// TIA Portal V19 program export: 1 tag tables, 127 data types, 0 data blocks, 65 code blocks (in call order from the OBs), 0 instance data blocks

VAR_GLOBAL   // PLC tag table "Parameterwaardes"
END_VAR
VAR_GLOBAL CONSTANT   // user constants
   Ja : USInt := 11;
   Aan : USInt := 12;
   Open : USInt := 13;
   Beschikbaar : USInt := 14;
   InDienst : USInt := 16;
   Bevestiging : USInt := 17;
   OK : USInt := 18;
   Geactiveerd : USInt := 19;
   Auto : USInt := 128;
   Manueel : USInt := 129;
   Hand : USInt := 130;
   Sensorregeling : USInt := 112;
   Uit : USInt := 42;
   Bereikt : USInt := 15;
   Beperkt : USInt := 21;
   Gedeeltelijk : USInt := 22;
   InTransitie : USInt := 23;
   OpenVerlaten : USInt := 24;
   DeelsAfgesloten : USInt := 25;
   Onbepaald : USInt := 26;
   Nee : USInt := 41;
   Dicht : USInt := 43;
   NietBeschikbaar : USInt := 44;
   Storing : USInt := 45;
   OnvoorwaardelijkDicht : USInt := 46;
   Geen : USInt := 47;
   UitDienst : USInt := 48;
   Annulering : USInt := 49;
   Fout : USInt := 50;
   NietBereikt : USInt := 51;
   Onderdrukt : USInt := 52;
   Stop : USInt := 53;
   Overbrugd : USInt := 54;
   NOK : USInt := 55;
   Gedeactiveerd : USInt := 56;
   Gedoofd : USInt := 61;
   Rood : USInt := 62;
   GeelKnipper : USInt := 63;
   Geel : USInt := 64;
   Groen : USInt := 65;
   Leeg : USInt := 70;
   LLW : USInt := 71;
   LW : USInt := 72;
   SW : USInt := 73;
   MSW : USInt := 74;
   LHW : USInt := 75;
   HHW : USInt := 76;
   Rijrichting : USInt := 81;
   Hoog : USInt := 82;
   Max : USInt := 83;
   Gent : USInt := 84;
   Oplopend : USInt := 85;
   Dag : USInt := 86;
   Tegenrij : USInt := 91;
   Laag : USInt := 92;
   Min : USInt := 93;
   Luik : USInt := 94;
   Aflopend : USInt := 95;
   Nacht : USInt := 96;
   Lokaal : USInt := 101;
   Centraal : USInt := 102;
   Licht : USInt := 105;
   Matig : USInt := 106;
   Waarneembaar : USInt := 107;
   Ernstig : USInt := 108;
   Regeling : USInt := 111;
   Windmeting : USInt := 113;
   Bewaken : USInt := 115;
   Blussen : USInt := 116;
   Testen : USInt := 117;
   Klein : USInt := 120;
   Groot : USInt := 121;
   NietSel : USInt := 125;
   SelHand : USInt := 126;
   SelAuto : USInt := 127;
   Reset : USInt := 135;
   Parallel : USInt := 137;
   Eiland : USInt := 138;
   Live : USInt := 140;
   Boodschap : USInt := 141;
   Radio : USInt := 142;
   Gesprek : USInt := 145;
   Wacht : USInt := 146;
   Aanvraag : USInt := 147;
   Recirculatie : USInt := 150;
   Bergen : USInt := 153;
   LeegHouden : USInt := 154;
   Lozen : USInt := 155;
   OnderWater : USInt := 157;
   BovenWater : USInt := 158;
   Onderhoud : USInt := 160;
   Normaal : USInt := 161;
   Calamiteit : USInt := 162;
   StandBy : USInt := 163;
   Ondersteunend : USInt := 164;
   Evacuatie : USInt := 165;
   Vlucht : USInt := 166;
   Brand : USInt := 167;
   Waarschuw : USInt := 168;
   "TSCT+GL" : USInt := 200;   // Tunnelkoker van Gent naar Luik
   "TSCT+LG" : USInt := 201;   // Tunnelkoker van Luik naar Gent
   "TOKA+BR" : USInt := 202;   // Tunnelkoker van Brussel naar Rotterdam
   "TOKA+RB" : USInt := 203;   // Tunnelkoker van Rotterdam naar Brussel
   "TLUC+AR" : USInt := 204;   // Tunnelkoker van Antwerpen naar Rotterdam
   "TLUC+BA" : USInt := 205;   // Tunnelkoker van Brussel naar Antwerpen
   "TLUC+BR" : USInt := 206;   // Tunnelkoker van Brussel naar Rotterdam
   "TLUC+RA" : USInt := 207;   // Tunnelkoker van Rotterdam naar Antwerpen
   "TLUC+RB" : USInt := 208;   // Tunnelkoker van Rotterdam naar Brussel
   "TLUC+AB" : USInt := 209;   // Tunnelkoker van Antwerpen naar Brussel
   "TKZO+GR" : USInt := 210;   // Tunnelkoker van Gent naar Rotterdam
   "TKZO+RG" : USInt := 211;   // Tunnelkoker van Rotterdam naar Gent
   "TKZB+LG" : USInt := 212;   // Tunnelkoker van Luik naar Gent
   "TKZB+GL" : USInt := 213;   // Tunnelkoker van Gent naar Luik
   "TSCH+BR" : USInt := 214;   // Tunnelkoker van Brussel naar Rotterdam
   "TSCH+RB" : USInt := 215;   // Tunnelkoker van Rotterdam naar Brussel
   "TKZO+RA" : USInt := 216;   // Uitrit van Rotterdam naar Antwerpen
   "TKZO+AR" : USInt := 217;   // Inrit van Antwerpen naar Rotterdam
   "TKZB+KA" : USInt := 218;   // Uitrit kanalzone knooppunt naar Antwerpen
   "TKZB+LK" : USInt := 219;   // Uitrit luik naar kanaalzone knooppunt
   "TKZB+AK" : USInt := 220;   // Inrit antwerpen naar kanaalzone knooppunt
   "TKZB+KL" : USInt := 221;   // Inrit kanaalzone knooppunt naar Luik
END_VAR

TYPE "C205_VAR_IF_GVL_TYPIC"
   STRUCT
      BMO_AAN { ExternalAccessible := 'False'; ExternalVisible := 'False'; ExternalWritable := 'False'} : Bool;   // Geleideverlichting aan
      EXT_AUT { ExternalAccessible := 'False'; ExternalVisible := 'False'; ExternalWritable := 'False'} : Bool;   // Externe (hoofd) beveiliging aangesproken
      EXT_HW { ExternalAccessible := 'False'; ExternalVisible := 'False'; ExternalWritable := 'False'} : Bool;   // Sturings hardware (PLC) in storing
      STO { ExternalAccessible := 'False'; ExternalVisible := 'False'; ExternalWritable := 'False'} : Struct   // Opsomming van alle storingen en meldingen
         A001 : Bool;   // Beveiliging aangesproken
         A002 : Bool;   // Storing voeding geleideverlichting
         AT01 : Bool;   // Foute terugmelding: Geleideverlichting aangestuurd, terugmelding Aan niet (of te laat) ontvangen
         AT02 : Bool;   // Foute terugmelding: Geleideverlichting niet aangestuurd, terugmelding Aan blijft aanwezig
      END_STRUCT;
   END_STRUCT;
END_TYPE

TYPE "C701_STU_IF_KMI_TYPIC"
   STRUCT
      CMD_NORM { ExternalAccessible := 'False'; ExternalVisible := 'False'; ExternalWritable := 'False'} : Bool;   // Aansturing klimaatregeling in stand Normaal (1 = Aan)
      CMD_CIR { ExternalAccessible := 'False'; ExternalVisible := 'False'; ExternalWritable := 'False'} : Bool;   // Aansturing klimaatregeling in stand Recirculatie (1 = Aan)
   END_STRUCT;
END_TYPE

TYPE "C701_VAR_IF_DEX_TYPIC"
   STRUCT
      TME_HOOG { ExternalAccessible := 'False'; ExternalVisible := 'False'; ExternalWritable := 'False'} : Bool;   // Ruimtetemperatuur te hoog
      STO { ExternalAccessible := 'False'; ExternalVisible := 'False'; ExternalWritable := 'False'} : Bool;   // Storing algemeen dakextractor
   END_STRUCT;
END_TYPE

TYPE "C701_VAR_IF_DFU_TYPIC"
   STRUCT
      REQ_VE { ExternalAccessible := 'False'; ExternalVisible := 'False'; ExternalWritable := 'False'} : Bool;   // Warmtevraag
      REQ_KO { ExternalAccessible := 'False'; ExternalVisible := 'False'; ExternalWritable := 'False'} : Bool;   // Koudevraag
      TME_HOLA { ExternalAccessible := 'False'; ExternalVisible := 'False'; ExternalWritable := 'False'} : Bool;   // Ruimtetemperatuur te hoog of te laag
      STO { ExternalAccessible := 'False'; ExternalVisible := 'False'; ExternalWritable := 'False'} : Bool;   // Storing algemeen klimaatkast
   END_STRUCT;
END_TYPE

TYPE "C701_VAR_IF_KLB_TYPIC"
   STRUCT
      KLB_TOE { ExternalAccessible := 'False'; ExternalVisible := 'False'; ExternalWritable := 'False'} : Bool;   // Brandklep gesloten
   END_STRUCT;
END_TYPE

TYPE "C701_VAR_IF_KMI_TYPIC"
   STRUCT
      EXT_AUT { ExternalAccessible := 'False'; ExternalVisible := 'False'; ExternalWritable := 'False'} : Bool;   // Externe (hoofd) beveiliging aangesproken
      EXT_HW { ExternalAccessible := 'False'; ExternalVisible := 'False'; ExternalWritable := 'False'} : Bool;   // Sturings hardware (PLC) in storing
      STO { ExternalAccessible := 'False'; ExternalVisible := 'False'; ExternalWritable := 'False'} : Struct   // Opsomming van alle storingen en meldingen
         A001 : Bool;   // Storing algemeen luchtbehandelingssysteem
         A002 : Bool;   // Storing algemeen koelmachine
         A003 : Bool;   // Storing algemeen warmtepomp
         A004 : Bool;   // Storing brandklep gesloten
         A005 : Bool;   // Storing temperatuur besturingslokaal
         A006 : Bool;   // Storing algemeen besturingslokaal
         A007 : Bool;   // Storing temperatuur opleidings/trainer/test/pauze lokaal
         A008 : Bool;   // Storing algemeen opleidings/trainer/test/pauze lokaal
         A009 : Bool;   // Storing temperatuur vergaderzaal/kantoor
         A010 : Bool;   // Storing algemeen vergaderzaal/kantoor
         A011 : Bool;   // Storing temperatuur batterijlokaal
         A012 : Bool;   // Storing algemeen batterijlokaal
         A013 : Bool;   // Storing temperatuur astrid/gsm lokaal
         A014 : Bool;   // Storing algemeen astrid/gsm lokaal
         A015 : Bool;   // Storing temperatuur sanitaire ruimte
         A016 : Bool;   // Storing algemeen sanitaire ruimte
         AT01 : Bool;
         AT02 : Bool;
         M001 : Bool;
         M002 : Bool;
      END_STRUCT;
   END_STRUCT;
END_TYPE

TYPE "C701_VAR_IF_KMO_TYPIC"
   STRUCT
      STO { ExternalAccessible := 'False'; ExternalVisible := 'False'; ExternalWritable := 'False'} : Struct   // Opsomming van alle storingen
         A001 : Bool;   // Fout temperatuurmeting koelwater in
         A002 : Bool;   // Fout temperatuurmeting koelwater uit
         A003 : Bool;   // Fout drukmeting koelwater
         A004 : Bool;   // Fout flowmeting koelwater
         A005 : Bool;   // Fout algemeen koelmachine
         A006 : Bool;   // Fout circulatiepomp
      END_STRUCT;
   END_STRUCT;
END_TYPE

TYPE "C701_VAR_IF_KOKR_TYPIC"
   STRUCT
      STO { ExternalAccessible := 'False'; ExternalVisible := 'False'; ExternalWritable := 'False'} : Struct   // Opsomming van alle storingen
         A001 : Bool;   // Storing van de motorbeveiliging van pomp 1
         A002 : Bool;   // Storing van de motorbeveiliging van pomp 2
         A003 : Bool;   // Fout temperatuurmeting vertrek
         A004 : Bool;   // Fout temperatuurmeting retour
         A005 : Bool;   // Fout drukmeting
      END_STRUCT;
   END_STRUCT;
END_TYPE

TYPE "C701_VAR_IF_KVE_TYPIC"
   STRUCT
      TME_HOOG { ExternalAccessible := 'False'; ExternalVisible := 'False'; ExternalWritable := 'False'} : Bool;   // Ruimtetemperatuur te hoog
      STO { ExternalAccessible := 'False'; ExternalVisible := 'False'; ExternalWritable := 'False'} : Bool;   // Storing algemeen kanaalventilator
   END_STRUCT;
END_TYPE

TYPE "C701_VAR_IF_LBS_TYPIC"
   STRUCT
      WRE { ExternalAccessible := 'False'; ExternalVisible := 'False'; ExternalWritable := 'False'} : USInt;   // Werkingsregime
      BMO_HAND { ExternalAccessible := 'False'; ExternalVisible := 'False'; ExternalWritable := 'False'} : Bool;   // TRUE = Werkingsregime is handmatig ingesteld via lokale bediening
      "Vrijgave pomp verwarmingsbat" { ExternalAccessible := 'False'; ExternalVisible := 'False'; ExternalWritable := 'False'} : Bool;   // Gaat naar if verwarmingskring CHECKEN OF DEZE POMP NU HIER INZIT OF IN DE KRING
      REQ_VE { ExternalAccessible := 'False'; ExternalVisible := 'False'; ExternalWritable := 'False'} : Bool;   // Warmtevraag voor kring verwarmingsbatterijen
      REQ_KO { ExternalAccessible := 'False'; ExternalVisible := 'False'; ExternalWritable := 'False'} : Bool;   // Koelvraag voor kring koelbatterijen (luchtgroep)
      STO { ExternalAccessible := 'False'; ExternalVisible := 'False'; ExternalWritable := 'False'} : Struct   // Opsomming van alle storingen
         A001 : Bool;   // Storing van de motorbeveiliging van pulsie ventilator
         A002 : Bool;   // Storing van de motorbeveiliging van extractie ventilator
         A003 : Bool;   // Fout drukmeting pulsie
         A004 : Bool;   // Fout drukmeting extractie
         A005 : Bool;   // Fout temperatuurmeting pulsie
         A006 : Bool;   // Fout temperatuurmeting extractie
         A007 : Bool;   // Fout temperatuurmeting buitenlucht
         A008 : Bool;   // Antivries alarm
         A009 : Bool;   // Filter vuil verse lucht
         A010 : Bool;   // Filter vuil extractie lucht
         AT01 : Bool;   // Foute terugmelding: damper verse lucht aangestuurd, terugmelding niet (of te laat) ontvangen
         AT02 : Bool;   // Foute terugmelding: damper extractie lucht aangestuurd, terugmelding niet (of te laat) ontvangen
         M001 : Bool;   // De pulsie ventilator is afgekoppeld via de werkschakelaar
         M002 : Bool;   // De extractie ventilator is afgekoppeld via de werkschakelaar
      END_STRUCT;
   END_STRUCT;
END_TYPE

TYPE "C701_VAR_IF_VAT_BUF_TYPIC"
   STRUCT
      STO { ExternalAccessible := 'False'; ExternalVisible := 'False'; ExternalWritable := 'False'} : Struct   // Opsomming van alle storingen
         A001 : Bool;   // Fout temperatuurmeting in vertrek
         A002 : Bool;   // Fout temperatuurmeting uit vertrek
         A003 : Bool;   // Fout temperatuurmeting in retour
         A004 : Bool;   // Fout temperatuurmeting uit retour
      END_STRUCT;
   END_STRUCT;
END_TYPE

TYPE "C701_VAR_IF_VAT_TYPIC"
   STRUCT
      STO { ExternalAccessible := 'False'; ExternalVisible := 'False'; ExternalWritable := 'False'} : Struct   // Opsomming van alle storingen
         A001 : Bool;   // Alarm lage druk expansievat verwarming
         A002 : Bool;   // Fout drukmeting expansievat verwarming
         A003 : Bool;   // Alarm lage druk expansievat koeling
         A004 : Bool;   // Fout drukmeting expansievat koeling
      END_STRUCT;
   END_STRUCT;
END_TYPE

TYPE "C701_VAR_IF_VAV_TYPIC"
   STRUCT
      TME_HOOG { ExternalAccessible := 'False'; ExternalVisible := 'False'; ExternalWritable := 'False'} : Bool;   // Ruimtetemperatuur te hoog
      STO { ExternalAccessible := 'False'; ExternalVisible := 'False'; ExternalWritable := 'False'} : Bool;   // Storing algemeen VAV
   END_STRUCT;
END_TYPE

TYPE "C701_VAR_IF_VCO_TYPIC"
   STRUCT
      REQ_VE { ExternalAccessible := 'False'; ExternalVisible := 'False'; ExternalWritable := 'False'} : Bool;   // Warmtevraag
      REQ_KO { ExternalAccessible := 'False'; ExternalVisible := 'False'; ExternalWritable := 'False'} : Bool;   // Koelvraag
      TME_HOLA { ExternalAccessible := 'False'; ExternalVisible := 'False'; ExternalWritable := 'False'} : Bool;   // Ruimtetemperatuur te hoog of te laag
      STO { ExternalAccessible := 'False'; ExternalVisible := 'False'; ExternalWritable := 'False'} : Bool;   // Storing algemeen ventiloconvector
   END_STRUCT;
END_TYPE

TYPE "C701_VAR_IF_VEB_TYPIC"
   STRUCT
      REQ_VE { ExternalAccessible := 'False'; ExternalVisible := 'False'; ExternalWritable := 'False'} : Bool;   // Warmtevraag voor kring verwarmingsbatterijen
      STO { ExternalAccessible := 'False'; ExternalVisible := 'False'; ExternalWritable := 'False'} : Struct   // Opsomming van alle storingen
         A001 : Bool;   // Ruimtetemperatuur te laag
         A002 : Bool;   // Fout temperatuurmeting
      END_STRUCT;
   END_STRUCT;
END_TYPE

TYPE "C701_VAR_IF_VEKR_TYPIC"
   STRUCT
      STO { ExternalAccessible := 'False'; ExternalVisible := 'False'; ExternalWritable := 'False'} : Struct   // Opsomming van alle storingen
         A001 : Bool;   // Storing van de motorbeveiliging van de pomp
         A002 : Bool;   // Fout temperatuurmeting vertrek
         A003 : Bool;   // Fout temperatuurmeting retour
         A004 : Bool;   // Fout drukmeting
         M001 : Bool;   // De motor is afgekoppeld via de werkschakelaar
      END_STRUCT;
   END_STRUCT;
END_TYPE

TYPE "C701_VAR_IF_VNU_TYPIC"
   STRUCT
      STO { ExternalAccessible := 'False'; ExternalVisible := 'False'; ExternalWritable := 'False'} : Bool;   // Storing algemeen ventilatie unit
   END_STRUCT;
END_TYPE

TYPE "C701_VAR_IF_WMP_TYPIC"
   STRUCT
      REQ_KMO { ExternalAccessible := 'False'; ExternalVisible := 'False'; ExternalWritable := 'False'} : Bool;   // Vrijgave koelmachine bij te hoge koellast
      STO { ExternalAccessible := 'False'; ExternalVisible := 'False'; ExternalWritable := 'False'} : Bool;   // Storing algemeen warmtepomp
   END_STRUCT;
END_TYPE

TYPE "C701_VAR_KMI_TYPIC"
   STRUCT
      BST { ExternalAccessible := 'False'; ExternalVisible := 'False'; ExternalWritable := 'False'} : USInt;   // Bestuurbaarheid
   END_STRUCT;
END_TYPE

TYPE "C104_VAR_IF_NSA_TYPIC"
   STRUCT
      ENE { ExternalAccessible := 'False'; ExternalVisible := 'False'; ExternalWritable := 'False'} : Real;   // Geleverde energie per aggregaat [kWh]
      PHI { ExternalAccessible := 'False'; ExternalVisible := 'False'; ExternalWritable := 'False'} : Real;   // Fasehoek (cos phi)
      SPA1 { ExternalAccessible := 'False'; ExternalVisible := 'False'; ExternalWritable := 'False'} : Real;   // Spanningsniveau lijn 1
      SPA2 { ExternalAccessible := 'False'; ExternalVisible := 'False'; ExternalWritable := 'False'} : Real;   // Spanningsniveau lijn 2
      SPA3 { ExternalAccessible := 'False'; ExternalVisible := 'False'; ExternalWritable := 'False'} : Real;   // Spanningsniveau lijn 3
      STR { ExternalAccessible := 'False'; ExternalVisible := 'False'; ExternalWritable := 'False'} : Real;   // Stroomsterkte
      WRE { ExternalAccessible := 'False'; ExternalVisible := 'False'; ExternalWritable := 'False'} : Bool;   // TRUE = werkingsregime: Belast FALSE = werkingsregime: Onbelast
      STS1 { ExternalAccessible := 'False'; ExternalVisible := 'False'; ExternalWritable := 'False'} : Bool;   // Status: Standby
      STS2 { ExternalAccessible := 'False'; ExternalVisible := 'False'; ExternalWritable := 'False'} : Bool;   // Status: Storing
      STS3 { ExternalAccessible := 'False'; ExternalVisible := 'False'; ExternalWritable := 'False'} : Bool;   // Status: Uitgeschakeld
      STS4 { ExternalAccessible := 'False'; ExternalVisible := 'False'; ExternalWritable := 'False'} : Bool;   // Status: Test
      STS_AAN { ExternalAccessible := 'False'; ExternalVisible := 'False'; ExternalWritable := 'False'} : Bool;   // In bedrijf (AAN)
      LDE { ExternalAccessible := 'False'; ExternalVisible := 'False'; ExternalWritable := 'False'} : Bool;   // Lekdetectie NSA
      TYD_TOT_AAN_UUR { ExternalAccessible := 'False'; ExternalVisible := 'False'; ExternalWritable := 'False'} : LInt;   // TYD_TOT_AAN_UUR
      SNS { ExternalAccessible := 'False'; ExternalVisible := 'False'; ExternalWritable := 'False'} : Bool;   // Noodstop (1 = gedeactiveerd)
      OPT_LDE { ExternalAccessible := 'False'; ExternalVisible := 'False'; ExternalWritable := 'False'} : Bool;   // Lekdetectie brandstof dagtank
      OPT_NIV { ExternalAccessible := 'False'; ExternalVisible := 'False'; ExternalWritable := 'False'} : Real;   // Brandstof niveau brandstof dagtank
      OPT_HOOG { ExternalAccessible := 'False'; ExternalVisible := 'False'; ExternalWritable := 'False'} : Bool;   // Overvulbeveiliging brandstof dagtank aangesproken
      OPT_STO { ExternalAccessible := 'False'; ExternalVisible := 'False'; ExternalWritable := 'False'} : Bool;   // Dagtank noodstroomaggregaat in storing
      EXT_AUT { ExternalAccessible := 'False'; ExternalVisible := 'False'; ExternalWritable := 'False'} : Bool;   // Externe (hoofd) beveiliging aangesproken
      EXT_HW { ExternalAccessible := 'False'; ExternalVisible := 'False'; ExternalWritable := 'False'} : Bool;   // Sturings hardware (PLC) in storing
      STO { ExternalAccessible := 'False'; ExternalVisible := 'False'; ExternalWritable := 'False'} : Struct   // Opsomming van alle storingen
         A001 : Bool;   // Beveiliging aangesproken
         A002 : Bool;   // Noodstroomaggregaat in storing
         A003 : Bool;   // Algemene storing noodstroomaggregaat
         A004 : Bool;   // Lekdetectie NSA
         A005 : Bool;   // Noodstop van het noodstroomaggregaat is geactiveerd
         A006 : Bool;   // Dagtank noodstroomaggregaat in storing
         A007 : Bool;   // Lekdetectie brandstof dagtank
         A008 : Bool;   // Overvulbeveiliging brandstof dagtank aangesproken
      END_STRUCT;
   END_STRUCT;
END_TYPE

TYPE "C106_VAR_IF_HSI_TYPIC"
   STRUCT
      BSC1 { ExternalAccessible := 'False'; ExternalVisible := 'False'; ExternalWritable := 'False'} : Bool;   // Hoogspanningsinstallatie beschikbaar
      BSC2 { ExternalAccessible := 'False'; ExternalVisible := 'False'; ExternalWritable := 'False'} : Bool;   // Hoogspanningsinstallatie niet beschikbaar
      BSC3 { ExternalAccessible := 'False'; ExternalVisible := 'False'; ExternalWritable := 'False'} : Bool;   // Hoogspanningsinstallatie beperkt beschikbaar
      WRE1 { ExternalAccessible := 'False'; ExternalVisible := 'False'; ExternalWritable := 'False'} : Bool;   // Werkingsregime: Netbedrijf
      WRE2 { ExternalAccessible := 'False'; ExternalVisible := 'False'; ExternalWritable := 'False'} : Bool;   // Werkingsregime: Parallelbedrijf
      WRE3 { ExternalAccessible := 'False'; ExternalVisible := 'False'; ExternalWritable := 'False'} : Bool;   // Werkingsregime: Eilandbedrijf
      LUS_TOE { ExternalAccessible := 'False'; ExternalVisible := 'False'; ExternalWritable := 'False'} : Bool;   // Hoogspanningslus is gesloten
      EXT_AUT { ExternalAccessible := 'False'; ExternalVisible := 'False'; ExternalWritable := 'False'} : Bool;   // Externe (hoofd) beveiliging aangesproken
      EXT_HW { ExternalAccessible := 'False'; ExternalVisible := 'False'; ExternalWritable := 'False'} : Bool;   // Sturings hardware (PLC) in storing
      STO { ExternalAccessible := 'False'; ExternalVisible := 'False'; ExternalWritable := 'False'} : Struct   // Opsomming van alle storingen
         A001 : Bool;   // Beveiliging aangesproken
         A002 : Bool;   // Hoogspanningsinstallatie in storing
         A003 : Bool;   // Algemene storing hoogspanningsinstallatie
         A004 : Bool;   // Hoogspanningslus is geopend
      END_STRUCT;
   END_STRUCT;
END_TYPE

TYPE "C106_VAR_IF_MVI_TYPIC"
   STRUCT
      PWR1 { ExternalAccessible := 'False'; ExternalVisible := 'False'; ExternalWritable := 'False'} : Real;   // Geleverde actief vermogen per aggregaat
      PWR2 { ExternalAccessible := 'False'; ExternalVisible := 'False'; ExternalWritable := 'False'} : Real;   // Geleverde reactief vermogen per aggregaat
      SPA1 { ExternalAccessible := 'False'; ExternalVisible := 'False'; ExternalWritable := 'False'} : Real;   // Spanningsniveau lijn 1
      SPA2 { ExternalAccessible := 'False'; ExternalVisible := 'False'; ExternalWritable := 'False'} : Real;   // Spanningsniveau lijn 2
      SPA3 { ExternalAccessible := 'False'; ExternalVisible := 'False'; ExternalWritable := 'False'} : Real;   // Spanningsniveau lijn 3
      PSU_STO { ExternalAccessible := 'False'; ExternalVisible := 'False'; ExternalWritable := 'False'} : Bool;   // Storing door een fout op de UPS
      PSU_AUT { ExternalAccessible := 'False'; ExternalVisible := 'False'; ExternalWritable := 'False'} : Bool;   // Verzamelalarm actief: de beveiliging van de hulpvoeding is getript
      EXT_AUT { ExternalAccessible := 'False'; ExternalVisible := 'False'; ExternalWritable := 'False'} : Bool;   // Externe (hoofd) beveiliging aangesproken
      EXT_HW { ExternalAccessible := 'False'; ExternalVisible := 'False'; ExternalWritable := 'False'} : Bool;   // Sturings hardware (PLC) in storing
      STO { ExternalAccessible := 'False'; ExternalVisible := 'False'; ExternalWritable := 'False'} : Struct   // Opsomming van alle storingen
         A001 : Bool;   // Beveiliging aangesproken
         A002 : Bool;   // Hoogspanningsverdeelbord in storing
         A003 : Bool;   // Algemene storing hoogspanningsverdeelbord
         A004 : Bool;   // Alarm door een fout op de UPS
         A005 : Bool;   // Verzamelalarm actief: de beveiliging van de hulpvoeding is getript
      END_STRUCT;
   END_STRUCT;
END_TYPE

TYPE "C106_VAR_IF_NET_TYPIC"
   STRUCT
      BSC1 { ExternalAccessible := 'False'; ExternalVisible := 'False'; ExternalWritable := 'False'} : Bool;   // Netaansluiting beschikbaar
      BSC2 { ExternalAccessible := 'False'; ExternalVisible := 'False'; ExternalWritable := 'False'} : Bool;   // Netaansluiting niet beschikbaar
      BSC3 { ExternalAccessible := 'False'; ExternalVisible := 'False'; ExternalWritable := 'False'} : Bool;   // Netaansluiting beperkt beschikbaar
      STS_KR { ExternalAccessible := 'False'; ExternalVisible := 'False'; ExternalWritable := 'False'} : Bool;   // Kritiek
      STS_GKR { ExternalAccessible := 'False'; ExternalVisible := 'False'; ExternalWritable := 'False'} : Bool;   // Gestopt kritiek
      TYD_GKR { ExternalAccessible := 'False'; ExternalVisible := 'False'; ExternalWritable := 'False'} : Real;   // Tijdverloop voor Gestopt Kritiek
      EXT_AUT { ExternalAccessible := 'False'; ExternalVisible := 'False'; ExternalWritable := 'False'} : Bool;   // Externe (hoofd) beveiliging aangesproken
      EXT_HW { ExternalAccessible := 'False'; ExternalVisible := 'False'; ExternalWritable := 'False'} : Bool;   // Sturings hardware (PLC) in storing
      STO { ExternalAccessible := 'False'; ExternalVisible := 'False'; ExternalWritable := 'False'} : Struct   // Opsomming van alle storingen
         A001 : Bool;   // Beveiliging aangesproken
         A002 : Bool;   // Netaansluiting in storing
         A003 : Bool;   // Algemene storing netaansluiting
         A004 : Bool;   // Geen netaansluiting beschikbaar
         A005 : Bool;   // NSA niet gestart na uitval netaansluiting
      END_STRUCT;
   END_STRUCT;
END_TYPE

TYPE "C106_VAR_IF_NME_TYPIC"
   STRUCT
      BSC1 { ExternalAccessible := 'False'; ExternalVisible := 'False'; ExternalWritable := 'False'} : Bool;   // Transformator beschikbaar
      BSC2 { ExternalAccessible := 'False'; ExternalVisible := 'False'; ExternalWritable := 'False'} : Bool;   // Transformator niet beschikbaar
      BSC3 { ExternalAccessible := 'False'; ExternalVisible := 'False'; ExternalWritable := 'False'} : Bool;   // Transformator beperkt beschikbaar
      EXT_AUT { ExternalAccessible := 'False'; ExternalVisible := 'False'; ExternalWritable := 'False'} : Bool;   // Externe (hoofd) beveiliging aangesproken
      EXT_HW { ExternalAccessible := 'False'; ExternalVisible := 'False'; ExternalWritable := 'False'} : Bool;   // Sturings hardware (PLC) in storing
   END_STRUCT;
END_TYPE

TYPE "C106_VAR_IF_REL_TYPIC"
   STRUCT
      ALM { ExternalAccessible := 'False'; ExternalVisible := 'False'; ExternalWritable := 'False'} : Bool;   // Alarm per beveiligingsrelais per uitschakelbevel: TRUE = OK / FALSE = Alarm
      AUT_TOE { ExternalAccessible := 'False'; ExternalVisible := 'False'; ExternalWritable := 'False'} : Bool;   // Vermogenschakelaar TOE (gesloten)
      SCA_TOE { ExternalAccessible := 'False'; ExternalVisible := 'False'; ExternalWritable := 'False'} : Bool;   // Aardingschakelaar TOE (gesloten)
      SYNC { ExternalAccessible := 'False'; ExternalVisible := 'False'; ExternalWritable := 'False'} : Bool;   // Lijndifferentieel beveiligingsrelais loopt synchroon
      EXT_AUT { ExternalAccessible := 'False'; ExternalVisible := 'False'; ExternalWritable := 'False'} : Bool;   // Externe (hoofd) beveiliging aangesproken
      EXT_HW { ExternalAccessible := 'False'; ExternalVisible := 'False'; ExternalWritable := 'False'} : Bool;   // Sturings hardware (PLC) in storing
   END_STRUCT;
END_TYPE

TYPE "C106_VAR_REL_TYPIC"
   STRUCT
      AUT_STS { ExternalAccessible := 'False'; ExternalVisible := 'False'; ExternalWritable := 'False'} : USInt;   // Status van de vermogenschakelaar van de hoogspanning
   END_STRUCT;
END_TYPE

TYPE "C103_VAR_IF_HVI_TYPIC"
   STRUCT
      PWR1 { ExternalAccessible := 'False'; ExternalVisible := 'False'; ExternalWritable := 'False'} : Real;   // Actief vermogen
      PWR2 { ExternalAccessible := 'False'; ExternalVisible := 'False'; ExternalWritable := 'False'} : Real;   // Reactief vermogen
      SPA_1 { ExternalAccessible := 'False'; ExternalVisible := 'False'; ExternalWritable := 'False'} : Real;   // Spanningsniveau lijn 1
      SPA_2 { ExternalAccessible := 'False'; ExternalVisible := 'False'; ExternalWritable := 'False'} : Real;   // Spanningsniveau lijn 2
      SPA_3 { ExternalAccessible := 'False'; ExternalVisible := 'False'; ExternalWritable := 'False'} : Real;   // Spanningsniveau lijn 3
      SPA_4 { ExternalAccessible := 'False'; ExternalVisible := 'False'; ExternalWritable := 'False'} : Real;   // Lijnspanning L1-L2
      SPA_5 { ExternalAccessible := 'False'; ExternalVisible := 'False'; ExternalWritable := 'False'} : Real;   // Lijnspanning L2-L3
      SPA_6 { ExternalAccessible := 'False'; ExternalVisible := 'False'; ExternalWritable := 'False'} : Real;   // Lijnspanning L1-L3
      STR_1 { ExternalAccessible := 'False'; ExternalVisible := 'False'; ExternalWritable := 'False'} : Real;   // Stroom lijn 1
      STR_2 { ExternalAccessible := 'False'; ExternalVisible := 'False'; ExternalWritable := 'False'} : Real;   // Stroom lijn 2
      STR_3 { ExternalAccessible := 'False'; ExternalVisible := 'False'; ExternalWritable := 'False'} : Real;   // Stroom lijn 3
      STR_4 { ExternalAccessible := 'False'; ExternalVisible := 'False'; ExternalWritable := 'False'} : Real;   // Stroom nulleider
      PHI { ExternalAccessible := 'False'; ExternalVisible := 'False'; ExternalWritable := 'False'} : Real;   // Arbeidsfactor
      BEV_SPA { ExternalAccessible := 'False'; ExternalVisible := 'False'; ExternalWritable := 'False'} : Bool;   // Status beveiliging detectie railspanning
      SPA2 { ExternalAccessible := 'False'; ExternalVisible := 'False'; ExternalWritable := 'False'} : Bool;   // Status detectie railspanning
      SPA1_STO { ExternalAccessible := 'False'; ExternalVisible := 'False'; ExternalWritable := 'False'} : Bool;   // Status detectie railspanning
      PHI_OK { ExternalAccessible := 'False'; ExternalVisible := 'False'; ExternalWritable := 'False'} : Bool;   // Status fasebewaking
      HLP_OK { ExternalAccessible := 'False'; ExternalVisible := 'False'; ExternalWritable := 'False'} : Bool;   // Status hulpvoedingen (groepscontact)
      SPD_OK { ExternalAccessible := 'False'; ExternalVisible := 'False'; ExternalWritable := 'False'} : Bool;   // Status overspanningsbeveiliging
      SPA3_STO { ExternalAccessible := 'False'; ExternalVisible := 'False'; ExternalWritable := 'False'} : Bool;   // Status storing detectie railspanning
      SPA4_STO { ExternalAccessible := 'False'; ExternalVisible := 'False'; ExternalWritable := 'False'} : Bool;   // Status storing detectie railspanning
      STS1 { ExternalAccessible := 'False'; ExternalVisible := 'False'; ExternalWritable := 'False'} : Bool;   // Status van elke schuif [IN]
      STS2 { ExternalAccessible := 'False'; ExternalVisible := 'False'; ExternalWritable := 'False'} : Bool;   // Status van elke schuif [TEST]
      STS3 { ExternalAccessible := 'False'; ExternalVisible := 'False'; ExternalWritable := 'False'} : Bool;   // Status van elke schuif [UIT]
      AUT_TOE { ExternalAccessible := 'False'; ExternalVisible := 'False'; ExternalWritable := 'False'} : Bool;   // Standmelding van elke vermogenschakelaar TOE [gesloten]
      BEV_OK { ExternalAccessible := 'False'; ExternalVisible := 'False'; ExternalWritable := 'False'} : Bool;   // Standmelding beveiliging vertrek
   END_STRUCT;
END_TYPE

TYPE "C103_VAR_IF_HVN_TYPIC"
   STRUCT
      PWR1 { ExternalAccessible := 'False'; ExternalVisible := 'False'; ExternalWritable := 'False'} : Real;   // Actief vermogen
      PWR2 { ExternalAccessible := 'False'; ExternalVisible := 'False'; ExternalWritable := 'False'} : Real;   // Reactief vermogen
      SPA_1 { ExternalAccessible := 'False'; ExternalVisible := 'False'; ExternalWritable := 'False'} : Real;   // Spanningsniveau lijn 1
      SPA_2 { ExternalAccessible := 'False'; ExternalVisible := 'False'; ExternalWritable := 'False'} : Real;   // Spanningsniveau lijn 2
      SPA_3 { ExternalAccessible := 'False'; ExternalVisible := 'False'; ExternalWritable := 'False'} : Real;   // Spanningsniveau lijn 3
      SPA_4 { ExternalAccessible := 'False'; ExternalVisible := 'False'; ExternalWritable := 'False'} : Real;   // Lijnspanning L1-L2
      SPA_5 { ExternalAccessible := 'False'; ExternalVisible := 'False'; ExternalWritable := 'False'} : Real;   // Lijnspanning L2-L3
      SPA_6 { ExternalAccessible := 'False'; ExternalVisible := 'False'; ExternalWritable := 'False'} : Real;   // Lijnspanning L1-L3
      STR_1 { ExternalAccessible := 'False'; ExternalVisible := 'False'; ExternalWritable := 'False'} : Real;   // Stroom lijn 1
      STR_2 { ExternalAccessible := 'False'; ExternalVisible := 'False'; ExternalWritable := 'False'} : Real;   // Stroom lijn 2
      STR_3 { ExternalAccessible := 'False'; ExternalVisible := 'False'; ExternalWritable := 'False'} : Real;   // Stroom lijn 3
      STR_4 { ExternalAccessible := 'False'; ExternalVisible := 'False'; ExternalWritable := 'False'} : Real;   // Stroom nulleider
      PHI { ExternalAccessible := 'False'; ExternalVisible := 'False'; ExternalWritable := 'False'} : Real;   // Arbeidsfactor
      AUT_TOE { ExternalAccessible := 'False'; ExternalVisible := 'False'; ExternalWritable := 'False'} : Bool;   // Standmelding van elke vermogenschakelaar TOE [gesloten]
      SCL1 { ExternalAccessible := 'False'; ExternalVisible := 'False'; ExternalWritable := 'False'} : Bool;   // Standmelding externe bypass netspanning
      SCL2 { ExternalAccessible := 'False'; ExternalVisible := 'False'; ExternalWritable := 'False'} : Bool;   // Standmelding aankomstschakelaar UPS
   END_STRUCT;
END_TYPE

TYPE "C103_VAR_IF_OVB_TYPIC"
   STRUCT
      SCL { ExternalAccessible := 'False'; ExternalVisible := 'False'; ExternalWritable := 'False'} : Bool;   // Standmelding ingangszone 400V/230V
   END_STRUCT;
END_TYPE

TYPE "C103_VAR_IF_OVI_TYPIC"
   STRUCT
      SCL { ExternalAccessible := 'False'; ExternalVisible := 'False'; ExternalWritable := 'False'} : Bool;   // Standmelding aankomstschakelaar
   END_STRUCT;
END_TYPE

TYPE "C103_VAR_IF_OVN_TYPIC"
   STRUCT
      SCL1 { ExternalAccessible := 'False'; ExternalVisible := 'False'; ExternalWritable := 'False'} : Bool;   // Standmelding aankomstschakelaar normaal
      SCL2 { ExternalAccessible := 'False'; ExternalVisible := 'False'; ExternalWritable := 'False'} : Bool;   // Standmelding aankomstschakelaar no-break
      BEV { ExternalAccessible := 'False'; ExternalVisible := 'False'; ExternalWritable := 'False'} : Bool;   // Standmelding automaat kast verwarming en ventilatie
   END_STRUCT;
END_TYPE

TYPE "C104_VAR_IF_KLP_TYPIC"
   STRUCT
      OPEN { ExternalAccessible := 'False'; ExternalVisible := 'False'; ExternalWritable := 'False'} : Bool;   // Brandstofklep open
      TOE { ExternalAccessible := 'False'; ExternalVisible := 'False'; ExternalWritable := 'False'} : Bool;   // Brandstofklep dicht
      EXT_AUT { ExternalAccessible := 'False'; ExternalVisible := 'False'; ExternalWritable := 'False'} : Bool;   // Externe (hoofd) beveiliging aangesproken
      EXT_HW { ExternalAccessible := 'False'; ExternalVisible := 'False'; ExternalWritable := 'False'} : Bool;   // Sturings hardware (PLC) in storing
      STO { ExternalAccessible := 'False'; ExternalVisible := 'False'; ExternalWritable := 'False'} : Struct   // Opsomming van alle storingen
         A001 : Bool;   // Beveiliging aangesproken
         A002 : Bool;   // Brandstofklep in storing
         A003 : Bool;   // Algemene storing brandstofklep
      END_STRUCT;
   END_STRUCT;
END_TYPE

TYPE "C104_VAR_IF_NSI_TYPIC"
   STRUCT
      BSC1 { ExternalAccessible := 'False'; ExternalVisible := 'False'; ExternalWritable := 'False'} : Bool;   // Noodstroominstallatie beschikbaar
      BSC2 { ExternalAccessible := 'False'; ExternalVisible := 'False'; ExternalWritable := 'False'} : Bool;   // Noodstroominstallatie niet beschikbaar
      BSC3 { ExternalAccessible := 'False'; ExternalVisible := 'False'; ExternalWritable := 'False'} : Bool;   // Noodstroominstallatie beperkt beschikbaar
      ENE_TOT { ExternalAccessible := 'False'; ExternalVisible := 'False'; ExternalWritable := 'False'} : Real;   // Totaal energieverbruik noodstroominstallatie
   END_STRUCT;
END_TYPE

TYPE "C104_VAR_IF_OPT_TYPIC"
   STRUCT
      KLP_OPEN { ExternalAccessible := 'False'; ExternalVisible := 'False'; ExternalWritable := 'False'} : Bool;   // Kleppenregister open
      KLP_TOE { ExternalAccessible := 'False'; ExternalVisible := 'False'; ExternalWritable := 'False'} : Bool;   // Kleppenregister dicht
      VEN_AAN { ExternalAccessible := 'False'; ExternalVisible := 'False'; ExternalWritable := 'False'} : Bool;   // Ventilator aan
      EXT_AUT { ExternalAccessible := 'False'; ExternalVisible := 'False'; ExternalWritable := 'False'} : Bool;   // Externe (hoofd) beveiliging aangesproken
      EXT_HW { ExternalAccessible := 'False'; ExternalVisible := 'False'; ExternalWritable := 'False'} : Bool;   // Sturings hardware (PLC) in storing
      STO { ExternalAccessible := 'False'; ExternalVisible := 'False'; ExternalWritable := 'False'} : Struct   // Opsomming van alle storingen
         A001 : Bool;   // Beveiliging aangesproken
         A002 : Bool;   // Luchtbehandelingssysteem in storing
         A003 : Bool;   // Algemene storing luchtbehandelingssysteem
      END_STRUCT;
   END_STRUCT;
END_TYPE

TYPE "C104_VAR_IF_PMP_TYPIC"
   STRUCT
      AAN { ExternalAccessible := 'False'; ExternalVisible := 'False'; ExternalWritable := 'False'} : Bool;   // Brandstofpomp aan
      EXT_AUT { ExternalAccessible := 'False'; ExternalVisible := 'False'; ExternalWritable := 'False'} : Bool;   // Externe (hoofd) beveiliging aangesproken
      EXT_HW { ExternalAccessible := 'False'; ExternalVisible := 'False'; ExternalWritable := 'False'} : Bool;   // Sturings hardware (PLC) in storing
      STO { ExternalAccessible := 'False'; ExternalVisible := 'False'; ExternalWritable := 'False'} : Struct   // Opsomming van alle storingen
         A001 : Bool;   // Beveiliging aangesproken
         A002 : Bool;   // Brandstofpomp in storing
         A003 : Bool;   // Algemene storing brandstofpomp
      END_STRUCT;
   END_STRUCT;
END_TYPE

TYPE "C105_VAR_IF_UPS_TYPIC"
   STRUCT
      STS1 { ExternalAccessible := 'False'; ExternalVisible := 'False'; ExternalWritable := 'False'} : Bool;   // Status UPS [In batterijwerking]
      STS2 { ExternalAccessible := 'False'; ExternalVisible := 'False'; ExternalWritable := 'False'} : Bool;   // Status UPS [In bypass]
      STS3 { ExternalAccessible := 'False'; ExternalVisible := 'False'; ExternalWritable := 'False'} : Bool;   // Status UPS [In normale werking]
      TYD { ExternalAccessible := 'False'; ExternalVisible := 'False'; ExternalWritable := 'False'} : Time;   // Resterende autonomietijd [min]
      PWR { ExternalAccessible := 'False'; ExternalVisible := 'False'; ExternalWritable := 'False'} : Real;   // Resterend vermogen
      SPA1 { ExternalAccessible := 'False'; ExternalVisible := 'False'; ExternalWritable := 'False'} : Real;   // Uitgangsspanning 1
      SPA2 { ExternalAccessible := 'False'; ExternalVisible := 'False'; ExternalWritable := 'False'} : Real;   // Uitgangsspanning 2
      SPA3 { ExternalAccessible := 'False'; ExternalVisible := 'False'; ExternalWritable := 'False'} : Real;   // Uitgangsspanning 3
      STR1 { ExternalAccessible := 'False'; ExternalVisible := 'False'; ExternalWritable := 'False'} : Real;   // Uitgangsstroom 1
      STR2 { ExternalAccessible := 'False'; ExternalVisible := 'False'; ExternalWritable := 'False'} : Real;   // Uitgangsstroom 2
      STR3 { ExternalAccessible := 'False'; ExternalVisible := 'False'; ExternalWritable := 'False'} : Real;   // Uitgangsstroom 3
   END_STRUCT;
END_TYPE

TYPE "C201_STU_VLZ_TYPIC"
   STRUCT
      CMD { ExternalAccessible := 'False'; ExternalVisible := 'False'; ExternalWritable := 'False'} : USInt;   // Sturing verlichtingszone algemeen
   END_STRUCT;
END_TYPE

TYPE "C205_VAR_IF_AVE_TYPIC"
   STRUCT
      EXT_AUT { ExternalAccessible := 'False'; ExternalVisible := 'False'; ExternalWritable := 'False'} : Bool;   // Externe (hoofd) beveiliging aangesproken
      EXT_HW { ExternalAccessible := 'False'; ExternalVisible := 'False'; ExternalWritable := 'False'} : Bool;   // Sturings hardware (PLC) in storing
      STO { ExternalAccessible := 'False'; ExternalVisible := 'False'; ExternalWritable := 'False'} : Struct   // Opsomming van alle storingen en meldingen
         A001 : Bool;   // Beveiliging aangesproken
      END_STRUCT;
   END_STRUCT;
END_TYPE

TYPE "C205_VAR_IF_CVE_TYPIC"
   STRUCT
      EXT_AUT { ExternalAccessible := 'False'; ExternalVisible := 'False'; ExternalWritable := 'False'} : Bool;   // Externe (hoofd) beveiliging aangesproken
      EXT_HW { ExternalAccessible := 'False'; ExternalVisible := 'False'; ExternalWritable := 'False'} : Bool;   // Sturings hardware (PLC) in storing
      STO { ExternalAccessible := 'False'; ExternalVisible := 'False'; ExternalWritable := 'False'} : Struct   // Opsomming van alle storingen en meldingen
         A001 : Bool;   // Beveiliging aangesproken
         A002 : Bool;   // Storing batterij
      END_STRUCT;
   END_STRUCT;
END_TYPE

TYPE "C301_STU_CLUST_TYPIC"
   STRUCT
      CMD_CAPA_CAPA { ExternalAccessible := 'False'; ExternalVisible := 'False'; ExternalWritable := 'False'} : USInt;   // Sturing ventilatie algemeen
      CMD_DIR { ExternalAccessible := 'False'; ExternalVisible := 'False'; ExternalWritable := 'False'} : USInt;   // Sturing richting
      CMD_ONHD { ExternalAccessible := 'False'; ExternalVisible := 'False'; ExternalWritable := 'False'} : USInt;   // Cluster die automatische onderhoudstesten moet uitvoeren
      VGV_BEV { ExternalAccessible := 'False'; ExternalVisible := 'False'; ExternalWritable := 'False'} : USInt;   // Vrijgave ventilator-beveiligingen onbalans en temperatuur
   END_STRUCT;
END_TYPE

TYPE "C301_STU_IF_VEN_TYPIC"
   STRUCT
      CMD_POS { ExternalAccessible := 'False'; ExternalVisible := 'False'; ExternalWritable := 'False'} : Bool;   // Aansturing ventilator positieve richting (Rijrichting)
      CMD_NEG { ExternalAccessible := 'False'; ExternalVisible := 'False'; ExternalWritable := 'False'} : Bool;   // Aansturing ventilator negatieve richting (Tegenrij)
      CMD_RES { ExternalAccessible := 'False'; ExternalVisible := 'False'; ExternalWritable := 'False'} : Bool;   // Reset van de latched storingen
   END_STRUCT;
END_TYPE

TYPE "C301_STU_VEN_TYPIC"
   STRUCT
      CMD { ExternalAccessible := 'False'; ExternalVisible := 'False'; ExternalWritable := 'False'} : USInt;   // Sturing ventilator
      BST { ExternalAccessible := 'False'; ExternalVisible := 'False'; ExternalWritable := 'False'} : USInt;   // Sturing In dienst / Uit dienst
      VGV_BEV { ExternalAccessible := 'False'; ExternalVisible := 'False'; ExternalWritable := 'False'} : USInt;   // Vrijgave ventilator-beveiligingen onbalans en temperatuur
   END_STRUCT;
END_TYPE

TYPE "C301_VAR_CLUST_TYPIC"
   STRUCT
      CAPA_OK { ExternalAccessible := 'False'; ExternalVisible := 'False'; ExternalWritable := 'False'} : USInt;   // Aantal bestuurbare ventilatoren in de cluster
      NIV_AAN_BWA { ExternalAccessible := 'False'; ExternalVisible := 'False'; ExternalWritable := 'False'} : USInt;   // Aantal aangeschakelde ventilatoren in de gewenste ventilatierichting
      DIR { ExternalAccessible := 'False'; ExternalVisible := 'False'; ExternalWritable := 'False'} : USInt;   // Richting van de cluster
      BMO { ExternalAccessible := 'False'; ExternalVisible := 'False'; ExternalWritable := 'False'} : USInt;   // Bedieningsmode
      ONHD_STS { ExternalAccessible := 'False'; ExternalVisible := 'False'; ExternalWritable := 'False'} : USInt;   // Status automatische onderhoudstesten
      PWR { ExternalAccessible := 'False'; ExternalVisible := 'False'; ExternalWritable := 'False'} : Real;   // Actueel vermogen van de ventilatiecluster
   END_STRUCT;
END_TYPE

TYPE "C301_VAR_IF_VEN_TYPIC"
   STRUCT
      STS_AAN { ExternalAccessible := 'False'; ExternalVisible := 'False'; ExternalWritable := 'False'} : Bool;   // TRUE = Ventilator is aangestuurd FALSE = Uit
      DIR_POS { ExternalAccessible := 'False'; ExternalVisible := 'False'; ExternalWritable := 'False'} : Bool;   // TRUE = Ventilator draait in positieve richting (rijrichting)
      DIR_NEG { ExternalAccessible := 'False'; ExternalVisible := 'False'; ExternalWritable := 'False'} : Bool;   // TRUE = Ventilator draait in negatieve richting (tegenrij)
      BMO_HAND { ExternalAccessible := 'False'; ExternalVisible := 'False'; ExternalWritable := 'False'} : Bool;   // TRUE = Ventilator in hand geschakeld FALSE = niet in hand
      TYD_TOT_AAN { ExternalAccessible := 'False'; ExternalVisible := 'False'; ExternalWritable := 'False'} : LInt;   // Totaal aantal draaiuren
      TYD_TOT_AAN_UUR { ExternalAccessible := 'False'; ExternalVisible := 'False'; ExternalWritable := 'False'} : LInt;   // Totaal aantal draaiuren
      ENE_MWA1 { ExternalAccessible := 'False'; ExternalVisible := 'False'; ExternalWritable := 'False'} : Real;   // Stroommeting fase 1
      ENE_MWA2 { ExternalAccessible := 'False'; ExternalVisible := 'False'; ExternalWritable := 'False'} : Real;   // Stroommeting fase 2
      ENE_MWA3 { ExternalAccessible := 'False'; ExternalVisible := 'False'; ExternalWritable := 'False'} : Real;   // Stroommeting fase 3
      TRL_MWA { ExternalAccessible := 'False'; ExternalVisible := 'False'; ExternalWritable := 'False'} : Real;   // Trillingsmeting
      EXT_AUT { ExternalAccessible := 'False'; ExternalVisible := 'False'; ExternalWritable := 'False'} : Bool;   // Externe (hoofd) beveiliging aangesproken
      EXT_HW { ExternalAccessible := 'False'; ExternalVisible := 'False'; ExternalWritable := 'False'} : Bool;   // Sturings hardware (PLC) in storing
      STO { ExternalAccessible := 'False'; ExternalVisible := 'False'; ExternalWritable := 'False'} : Struct   // Opsomming van alle storingen en meldingen
         A001 : Bool;   // Beveiliging aangesproken
         A002 : Bool;   // Algemene storing MCC
         A003 : Bool;   // Te hoge temperatuur in de wikkelingen van de motor van de ventilator
         A004 : Bool;   // De ventilator is in onbalans
         A005 : Bool;   // Fout stroommeting fase 1
         A006 : Bool;   // Fout stroommeting fase 2
         A007 : Bool;   // Fout stroommeting fase 3
         A008 : Bool;   // Motorlade uitgeschakeld
         A009 : Bool;   // Motorlade in test
         A010 : Bool;   // Motorlade uitgereden
         A011 : Bool;   // Draadbreuk trillingsmeting
         A012 : Bool;   // Meetbereik trillingsmeting overschreden
         AT01 : Bool;   // Discordantie motor: terugmelding niet ontvangen
         AT02 : Bool;   // Discordantie motor: terugmelding blijft aanwezig
         AT03 : Bool;   // Discordantie motor: terugmeldingen Positief en negatief tegelijkertijd
         M001 : Bool;   // Werkschakelaar uitgeschakeld
      END_STRUCT;
   END_STRUCT;
END_TYPE

TYPE "C301_VAR_VEN_TYPIC"
   STRUCT
      STS { ExternalAccessible := 'False'; ExternalVisible := 'False'; ExternalWritable := 'False'} : USInt;   // Status van de ventilator
      DIR { ExternalAccessible := 'False'; ExternalVisible := 'False'; ExternalWritable := 'False'} : USInt;   // Richting van de ventilator
      BMO { ExternalAccessible := 'False'; ExternalVisible := 'False'; ExternalWritable := 'False'} : USInt;   // Bedieningsmode
      BST { ExternalAccessible := 'False'; ExternalVisible := 'False'; ExternalWritable := 'False'} : USInt;   // Bestuurbaarheid
      PWR { ExternalAccessible := 'False'; ExternalVisible := 'False'; ExternalWritable := 'False'} : Real;   // Vermogen van de ventilator
      TYD_TOT_AAN { ExternalAccessible := 'False'; ExternalVisible := 'False'; ExternalWritable := 'False'} : USInt;   // Totaal aantal draaiuren
   END_STRUCT;
END_TYPE

TYPE "C302_VAR_IF_LKM_TYPIC"
   STRUCT
      LKM_MWA { ExternalAccessible := 'False'; ExternalVisible := 'False'; ExternalWritable := 'False'} : Real;   // Meetwaarde [m-1]
      EXT_AUT { ExternalAccessible := 'False'; ExternalVisible := 'False'; ExternalWritable := 'False'} : Bool;   // Externe (hoofd) beveiliging aangesproken
      EXT_HW { ExternalAccessible := 'False'; ExternalVisible := 'False'; ExternalWritable := 'False'} : Bool;   // Sturings hardware (PLC) in storing
      STO { ExternalAccessible := 'False'; ExternalVisible := 'False'; ExternalWritable := 'False'} : Struct   // Opsomming van alle storingen
         A001 : Bool;   // Luchtkwaliteitsmeter niet aangeschakeld
         A002 : Bool;   // Draadbreuk analoge meting
         A003 : Bool;   // Meetbereik overschreden
         A004 : Bool;   // Luchtkwaliteitsmeter geeft storing
      END_STRUCT;
   END_STRUCT;
END_TYPE

TYPE "C302_VAR_LKM_TYPIC"
   STRUCT
      MWA { ExternalAccessible := 'False'; ExternalVisible := 'False'; ExternalWritable := 'False'} : USInt;   // Meetwaarde (uitgemiddelde k-waarde)
      POS { ExternalAccessible := 'False'; ExternalVisible := 'False'; ExternalWritable := 'False'} : USInt;   // Lengtepositie van de luchtkwaliteitsmeter in de verkeerskoker
      VAR_ROOK { ExternalAccessible := 'False'; ExternalVisible := 'False'; ExternalWritable := 'False'} : USInt;   // Rookdetectie
      OBS { ExternalAccessible := 'False'; ExternalVisible := 'False'; ExternalWritable := 'False'} : USInt;   // Observeerbaarheid
      NUM_VOOR { ExternalAccessible := 'False'; ExternalVisible := 'False'; ExternalWritable := 'False'} : Int;   // Nummer van de voorafgaande luchtkwaliteitsmeter
      NUM_NA { ExternalAccessible := 'False'; ExternalVisible := 'False'; ExternalWritable := 'False'} : Int;   // Nummer van de volgende luchtkwaliteitsmeter
   END_STRUCT;
END_TYPE

TYPE "C401_VAR_IF_RSS_TYPIC"
   STRUCT
      STS { ExternalAccessible := 'False'; ExternalVisible := 'False'; ExternalWritable := 'False'} : String[8];   // Naam van de getoonde beeldstand (bitmap) op het bord
      EXT_AUT { ExternalAccessible := 'False'; ExternalVisible := 'False'; ExternalWritable := 'False'} : Bool;   // Externe (hoofd) beveiliging aangesproken
      EXT_HW { ExternalAccessible := 'False'; ExternalVisible := 'False'; ExternalWritable := 'False'} : Bool;   // Sturings hardware (PLC) in storing
      STO { ExternalAccessible := 'False'; ExternalVisible := 'False'; ExternalWritable := 'False'} : Struct   // Opsomming van alle storingen en meldingen
         A001 : Bool;   // Beveiliging aangesproken
         A002 : Bool;   // Storing luspaar
         A003 : Bool;   // Storing RSS-bord gedetecteerd door PRTG
         A004 : Bool;   // Storing RSS-bord
         A005 : Bool;   // Algemene storing RSS-bord
      END_STRUCT;
   END_STRUCT;
END_TYPE

TYPE "C401_VAR_RSS_TYPIC"
   STRUCT
      OBS { ExternalAccessible := 'False'; ExternalVisible := 'False'; ExternalWritable := 'False'} : USInt;   // Observeerbaarheid
      LUS_STO { ExternalAccessible := 'False'; ExternalVisible := 'False'; ExternalWritable := 'False'} : USInt;   // Storingsstatus luspaar
   END_STRUCT;
END_TYPE

TYPE "C402_STU_AFS_IF_SBO_TYPIC"
   STRUCT
      CMD_HND { ExternalAccessible := 'False'; ExternalVisible := 'False'; ExternalWritable := 'False'} : Bool;   // Commando Bedieningsmode Hand activeren
      CMD_OPEN { ExternalAccessible := 'False'; ExternalVisible := 'False'; ExternalWritable := 'False'} : Bool;   // Commando Openen afsluitboom (voor hulpdiensten)
      STS_VKL_OK { ExternalAccessible := 'False'; ExternalVisible := 'False'; ExternalWritable := 'False'} : Bool;   // 1 = Verkeerslichten op Rood
      EXT_STO { ExternalAccessible := 'False'; ExternalVisible := 'False'; ExternalWritable := 'False'} : Bool;   // Externe storing aanwezig
      EXT_NDS_NOK { ExternalAccessible := 'False'; ExternalVisible := 'False'; ExternalWritable := 'False'} : Bool;   // Noodstopkring niet in orde
   END_STRUCT;
END_TYPE

TYPE "C402_STU_AFS_IF_VKL_TYPIC"
   STRUCT
      CMD_HND { ExternalAccessible := 'False'; ExternalVisible := 'False'; ExternalWritable := 'False'} : Bool;   // Commando Bedieningsmode Hand activeren
      CMD_HND_ROOD { ExternalAccessible := 'False'; ExternalVisible := 'False'; ExternalWritable := 'False'} : Bool;   // Handmatig commando Rood
      CMD_HND_GROE { ExternalAccessible := 'False'; ExternalVisible := 'False'; ExternalWritable := 'False'} : Bool;   // Handmatig commando Groen
      CMD_HND_KNIP { ExternalAccessible := 'False'; ExternalVisible := 'False'; ExternalWritable := 'False'} : Bool;   // Handmatig commando Geel Knipperen
      CMD_HND_UIT { ExternalAccessible := 'False'; ExternalVisible := 'False'; ExternalWritable := 'False'} : Bool;   // Handmatig commando Uit
      STO_ROOD { ExternalAccessible := 'False'; ExternalVisible := 'False'; ExternalWritable := 'False'} : Bool;   // Geen enkel verkeerslicht kan de stand rood tonen
   END_STRUCT;
END_TYPE

TYPE "C402_STU_IF_AFS_TYPIC"
   STRUCT
      STU_RES { ExternalAccessible := 'False'; ExternalVisible := 'False'; ExternalWritable := 'False'} : Bool;   // True = reset noodstop kring False = geen sturing
   END_STRUCT;
END_TYPE

TYPE "C402_STU_IF_M33_TYPIC"
   STRUCT
      CMD_AAN { ExternalAccessible := 'False'; ExternalVisible := 'False'; ExternalWritable := 'False'} : Bool;   // TRUE = weergeven beeldstand verkeerslicht FALSE = niets weergeven
      CMD_RES { ExternalAccessible := 'False'; ExternalVisible := 'False'; ExternalWritable := 'False'} : Bool;   // Reset van de latched storingen
   END_STRUCT;
END_TYPE

TYPE "C402_STU_IF_SBO_TYPIC"
   STRUCT
      CMD_OPEN { ExternalAccessible := 'False'; ExternalVisible := 'False'; ExternalWritable := 'False'} : Bool;   // Aansturing afsluitboom Open
      CMD_VWA_TOE { ExternalAccessible := 'False'; ExternalVisible := 'False'; ExternalWritable := 'False'} : Bool;   // Aansturing afsluitboom voorwaardelijk Dicht
      CMD_TOE { ExternalAccessible := 'False'; ExternalVisible := 'False'; ExternalWritable := 'False'} : Bool;   // Aansturing afsluitboom (onvoorwaardelijk) Dicht
      CMD_STOP { ExternalAccessible := 'False'; ExternalVisible := 'False'; ExternalWritable := 'False'} : Bool;   // Aansturing afsluitboom Stop
      CMD_RES { ExternalAccessible := 'False'; ExternalVisible := 'False'; ExternalWritable := 'False'} : Bool;   // Reset van de latched storingen
      VGV_SNEL { ExternalAccessible := 'False'; ExternalVisible := 'False'; ExternalWritable := 'False'} : Bool;   // Vrijgave om versneld te sluiten
   END_STRUCT;
END_TYPE

TYPE "C402_STU_IF_VKL_TYPIC"
   STRUCT
      COMM_OK { ExternalAccessible := 'False'; ExternalVisible := 'False'; ExternalWritable := 'False'} : Bool;   // Communicatie met 3B in werking
      CMD_ROOD { ExternalAccessible := 'False'; ExternalVisible := 'False'; ExternalWritable := 'False'} : Bool;   // Aansturing verkeerslicht Rood
      CMD_GROE { ExternalAccessible := 'False'; ExternalVisible := 'False'; ExternalWritable := 'False'} : Bool;   // Aansturing verkeerslicht Groen
      CMD_KNIP { ExternalAccessible := 'False'; ExternalVisible := 'False'; ExternalWritable := 'False'} : Bool;   // Aansturing verkeerslicht Geel Knipperen
      CMD_RES { ExternalAccessible := 'False'; ExternalVisible := 'False'; ExternalWritable := 'False'} : Bool;   // Reset van de latched storingen
      CMD_ONHD { ExternalAccessible := 'False'; ExternalVisible := 'False'; ExternalWritable := 'False'} : Bool;   // Automatische onderhoudstesten uitvoeren
      VGV_SNEL { ExternalAccessible := 'False'; ExternalVisible := 'False'; ExternalWritable := 'False'} : Bool;   // Vrijgave om versneld naar rood te gaan
   END_STRUCT;
END_TYPE

TYPE "C402_STU_M33_TYPIC"
   STRUCT
      CMD { ExternalAccessible := 'False'; ExternalVisible := 'False'; ExternalWritable := 'False'} : Bool;   // Sturing M33-bord
   END_STRUCT;
END_TYPE

TYPE "C402_STU_SBO_TYPIC"
   STRUCT
      CMD { ExternalAccessible := 'False'; ExternalVisible := 'False'; ExternalWritable := 'False'} : USInt;   // Sturing positionering afsluitboom
      SNEL { ExternalAccessible := 'False'; ExternalVisible := 'False'; ExternalWritable := 'False'} : USInt;   // Sturing versneld
      VGV_TOE { ExternalAccessible := 'False'; ExternalVisible := 'False'; ExternalWritable := 'False'} : USInt;   // Vrijgave sluiten (verkeerslichten voldoende lang op Rood)
      VGV_VWA_TOE { ExternalAccessible := 'False'; ExternalVisible := 'False'; ExternalWritable := 'False'} : USInt;   // Vrijgave voorwaardelijk sluiten
   END_STRUCT;
END_TYPE

TYPE "C402_STU_VKL_TYPIC"
   STRUCT
      CMD { ExternalAccessible := 'False'; ExternalVisible := 'False'; ExternalWritable := 'False'} : USInt;   // Sturing verkeerslicht
      CMD_ONHD { ExternalAccessible := 'False'; ExternalVisible := 'False'; ExternalWritable := 'False'} : USInt;   // Automatische onderhoudstesten uitvoeren
      SNEL { ExternalAccessible := 'False'; ExternalVisible := 'False'; ExternalWritable := 'False'} : USInt;   // Sturing versneld
   END_STRUCT;
END_TYPE

TYPE "C402_VAR_IF_AFS_TYPIC"
   STRUCT
      STS_VKL_OK { ExternalAccessible := 'False'; ExternalVisible := 'False'; ExternalWritable := 'False'} : Bool;   // TRUE = verkeerslichten op rood, vrijgave sluiten afsluitbomen
      STS_VKL_AAN { ExternalAccessible := 'False'; ExternalVisible := 'False'; ExternalWritable := 'False'} : Bool;   // TRUE = verkeerslichten aangestuurd
      STS_KST_OPEN { ExternalAccessible := 'False'; ExternalVisible := 'False'; ExternalWritable := 'False'} : Bool;   // TRUE = deur wegkantkast geopend
      STO { ExternalAccessible := 'False'; ExternalVisible := 'False'; ExternalWritable := 'False'} : Struct   // Opsomming van alle signaleringen
         A001 : Bool;   // Noodstop
         A002 : Bool;   // Storing UPS
         A003 : Bool;   // UPS in batterijwerking
         A004 : Bool;   // Storing klimaatregeling wegkantkast
      END_STRUCT;
   END_STRUCT;
END_TYPE

TYPE "C402_VAR_IF_M33_TYPIC"
   STRUCT
      STS_AAN { ExternalAccessible := 'False'; ExternalVisible := 'False'; ExternalWritable := 'False'} : Bool;   // TRUE = M33-bord actueel in werking FALSE = Uit
      EXT_AUT { ExternalAccessible := 'False'; ExternalVisible := 'False'; ExternalWritable := 'False'} : Bool;   // Externe (hoofd) beveiliging aangesproken
      EXT_HW { ExternalAccessible := 'False'; ExternalVisible := 'False'; ExternalWritable := 'False'} : Bool;   // Sturings hardware (PLC) in storing
      STO { ExternalAccessible := 'False'; ExternalVisible := 'False'; ExternalWritable := 'False'} : Struct   // Opsomming van alle storingen en meldingen
         A001 : Bool;   // Beveiliging aangesproken
         A002 : Bool;   // Storing M33-bord gedetecteerd door PRTG
         A003 : Bool;   // Storing M33-bord
         A004 : Bool;   // Algemene storing M33-bord
         AT01 : Bool;   // Foute terugmelding: M33-bord aangestuurd, terugmelding Aan niet (of te laat) ontvangen
         AT02 : Bool;   // Foute terugmelding: M33-bord niet aangestuurd, terugmelding Aan blijft aanwezig
      END_STRUCT;
   END_STRUCT;
END_TYPE

TYPE "C402_VAR_IF_SBO_TYPIC"
   STRUCT
      STS_BEZ_OPEN { ExternalAccessible := 'False'; ExternalVisible := 'False'; ExternalWritable := 'False'} : Bool;   // TRUE = Afsluitboom bezig met beweging openen
      STS_BEZ_TOE { ExternalAccessible := 'False'; ExternalVisible := 'False'; ExternalWritable := 'False'} : Bool;   // TRUE = Afsluitboom bezig met beweging sluiten
      STS_OPEN { ExternalAccessible := 'False'; ExternalVisible := 'False'; ExternalWritable := 'False'} : Bool;   // TRUE = Afsluitboom op stand Open
      STS_TOE { ExternalAccessible := 'False'; ExternalVisible := 'False'; ExternalWritable := 'False'} : Bool;   // TRUE = Afsluitboom op stand Dicht
      STS_STOP { ExternalAccessible := 'False'; ExternalVisible := 'False'; ExternalWritable := 'False'} : Bool;   // TRUE = Afsluitboom niet op een eindpositie en niet in beweging
      BMO_HAND { ExternalAccessible := 'False'; ExternalVisible := 'False'; ExternalWritable := 'False'} : Bool;   // TRUE = Afsluitboom in hand geschakeld / FALSE = niet in hand
      STS_VKL_OK { ExternalAccessible := 'False'; ExternalVisible := 'False'; ExternalWritable := 'False'} : Bool;   // TRUE = Verkeerslichten op Rood (voorwaarde voor sluiten)
      STS_NDS_OK { ExternalAccessible := 'False'; ExternalVisible := 'False'; ExternalWritable := 'False'} : Bool;   // TRUE = Geen noodstop (voorwaarde voor beweging)
      STS_LUS_OK { ExternalAccessible := 'False'; ExternalVisible := 'False'; ExternalWritable := 'False'} : Bool;   // TRUE = Detectielus(sen) OK (geen obstakel gedetecteerd voor sluiten)
      EXT_AUT { ExternalAccessible := 'False'; ExternalVisible := 'False'; ExternalWritable := 'False'} : Bool;   // Externe (hoofd) beveiliging aangesproken
      EXT_HW { ExternalAccessible := 'False'; ExternalVisible := 'False'; ExternalWritable := 'False'} : Bool;   // Sturings hardware (PLC) in storing
      EXT_STO { ExternalAccessible := 'False'; ExternalVisible := 'False'; ExternalWritable := 'False'} : Bool;   // Externe storing aanwezig
      LUS1_STS { ExternalAccessible := 'False'; ExternalVisible := 'False'; ExternalWritable := 'False'} : Bool;   // Detectie voertuig door lus 1 (1 = detectie)
      LUS2_STS { ExternalAccessible := 'False'; ExternalVisible := 'False'; ExternalWritable := 'False'} : Bool;   // Detectie voertuig door lus 2 (1 = detectie)
      LUS3_STS { ExternalAccessible := 'False'; ExternalVisible := 'False'; ExternalWritable := 'False'} : Bool;   // Detectie voertuig door lus 3 (1 = detectie)
      LUS4_STS { ExternalAccessible := 'False'; ExternalVisible := 'False'; ExternalWritable := 'False'} : Bool;   // Detectie voertuig door lus 3 (1 = detectie)
      STO { ExternalAccessible := 'False'; ExternalVisible := 'False'; ExternalWritable := 'False'} : Struct   // Opsomming van alle storingen
         A001 : Bool;   // Beveiliging aangesproken
         A002 : Bool;   // Storing van de detector van lus 1
         A003 : Bool;   // Storing van de detector van lus 2
         A004 : Bool;   // Storing van de detector van lus 3
         A005 : Bool;   // Storing van de detector van lus 4
         A006 : Bool;   // Storing van de motorsturing
         A007 : Bool;   // Storing motorbeveiliging
         AT01 : Bool;   // Terugmelding Open niet tijdig bereikt
         AT02 : Bool;   // Terugmelding Dicht niet tijdig bereikt
         AT03 : Bool;   // Terugmeldingen Open en Dicht tegelijkertijd
         AT04 : Bool;   // Terugmelding Open weggevallen
         AT05 : Bool;   // Terugmelding Dicht weggevallen
         M001 : Bool;   // Werkschakelaar uitgeschakeld
         M002 : Bool;   // Mechanische handbediening uitgenomen
      END_STRUCT;
   END_STRUCT;
END_TYPE

TYPE "C402_VAR_IF_VKL_TYPIC"
   STRUCT
      STS_ROOD { ExternalAccessible := 'False'; ExternalVisible := 'False'; ExternalWritable := 'False'} : Bool;   // TRUE = Verkeerslicht actueel op rood
      STS_GEEL { ExternalAccessible := 'False'; ExternalVisible := 'False'; ExternalWritable := 'False'} : Bool;   // TRUE = Verkeerslicht actueel op geel (vast)
      STS_GROE { ExternalAccessible := 'False'; ExternalVisible := 'False'; ExternalWritable := 'False'} : Bool;   // TRUE = Verkeerslicht actueel op groen
      STS_KNIP { ExternalAccessible := 'False'; ExternalVisible := 'False'; ExternalWritable := 'False'} : Bool;   // TRUE = Verkeerslicht actueel op knipperen geel
      STS_AAN { ExternalAccessible := 'False'; ExternalVisible := 'False'; ExternalWritable := 'False'} : Bool;   // TRUE = Verkeerslicht wordt aangestuurd
      BMO_HAND { ExternalAccessible := 'False'; ExternalVisible := 'False'; ExternalWritable := 'False'} : Bool;   // TRUE = Verkeerslicht in hand geschakeld / FALSE = niet in hand
      EXT_AUT { ExternalAccessible := 'False'; ExternalVisible := 'False'; ExternalWritable := 'False'} : Bool;   // Externe (hoofd) beveiliging aangesproken
      EXT_HW { ExternalAccessible := 'False'; ExternalVisible := 'False'; ExternalWritable := 'False'} : Bool;   // Sturings hardware (PLC) in storing
      STO { ExternalAccessible := 'False'; ExternalVisible := 'False'; ExternalWritable := 'False'} : Struct   // Opsomming van alle signaleringen
         A001 : Bool;   // Beveiliging aangesproken
         AT01 : Bool;   // De rode lens is defect
         AT02 : Bool;   // De gele lens is defect
         AT03 : Bool;   // De groene lens is defect
         AT04 : Bool;   // De stand rood kan niet getoond worden
         AT05 : Bool;   // De stand geel kan niet getoond worden
         AT06 : Bool;   // De stand geel knipperen kan niet getoond worden
         AT07 : Bool;   // De stand groen kan niet getoond worden
      END_STRUCT;
   END_STRUCT;
END_TYPE

TYPE "C402_VAR_M33_TYPIC"
   STRUCT
      STS { ExternalAccessible := 'False'; ExternalVisible := 'False'; ExternalWritable := 'False'} : USInt;   // Actuele status van het M33-bord
      BMO { ExternalAccessible := 'False'; ExternalVisible := 'False'; ExternalWritable := 'False'} : USInt;   // Bedieningsmode
      BST { ExternalAccessible := 'False'; ExternalVisible := 'False'; ExternalWritable := 'False'} : USInt;   // Bestuurbaarheid
   END_STRUCT;
END_TYPE

TYPE "C402_VAR_SBO_TYPIC"
   STRUCT
      BEZ_STS { ExternalAccessible := 'False'; ExternalVisible := 'False'; ExternalWritable := 'False'} : USInt;   // Status van de beweging van de afsluitboom
      POS_STS { ExternalAccessible := 'False'; ExternalVisible := 'False'; ExternalWritable := 'False'} : USInt;   // Status van de positie van de afsluitboom
      BMO { ExternalAccessible := 'False'; ExternalVisible := 'False'; ExternalWritable := 'False'} : USInt;   // Bedieningsmode
      BST { ExternalAccessible := 'False'; ExternalVisible := 'False'; ExternalWritable := 'False'} : USInt;   // Bestuurbaarheid
   END_STRUCT;
END_TYPE

TYPE "C402_VAR_VKL_TYPIC"
   STRUCT
      STS { ExternalAccessible := 'False'; ExternalVisible := 'False'; ExternalWritable := 'False'} : USInt;   // Actuele status van het verkeerslicht
      BMO { ExternalAccessible := 'False'; ExternalVisible := 'False'; ExternalWritable := 'False'} : USInt;   // Bedieningsmode
      BST { ExternalAccessible := 'False'; ExternalVisible := 'False'; ExternalWritable := 'False'} : USInt;   // Bestuurbaarheid
   END_STRUCT;
END_TYPE

TYPE "C403_STU_LVE_TYPIC"
   STRUCT
      LCK_STOP { ExternalAccessible := 'False'; ExternalVisible := 'False'; ExternalWritable := 'False'} : Array[1..7, 0..40] of Int;   // Lijst van detectiepunten die een stilstand signaleren
      LCK_SOS { ExternalAccessible := 'False'; ExternalVisible := 'False'; ExternalWritable := 'False'} : Array[1..7, 0..40] of Int;   // Lijst van detectiepunten die een snelheidsonderschrijding signaleren
      LCK_NEG { ExternalAccessible := 'False'; ExternalVisible := 'False'; ExternalWritable := 'False'} : USInt;   // Ja = Spookrijder detectie vergrendeld (niet actief)
   END_STRUCT;
END_TYPE

TYPE "C403_VAR_IF_LVE_TYPIC"
   STRUCT
      EXT_HW { ExternalAccessible := 'False'; ExternalVisible := 'False'; ExternalWritable := 'False'} : Bool;   // Sturings hardware (PLC) in storing
      STS_KST_OPEN { ExternalAccessible := 'False'; ExternalVisible := 'False'; ExternalWritable := 'False'} : Bool;   // TRUE = deur wegkantkast geopend
      STS_NEG { ExternalAccessible := 'False'; ExternalVisible := 'False'; ExternalWritable := 'False'} : Bool;   // Spookrijder gedetecteerd
      STS_SOS { ExternalAccessible := 'False'; ExternalVisible := 'False'; ExternalWritable := 'False'} : Bool;   // Snelheidsonderschrijding
      STS_STOP { ExternalAccessible := 'False'; ExternalVisible := 'False'; ExternalWritable := 'False'} : Bool;   // Stilstand
      STO { ExternalAccessible := 'False'; ExternalVisible := 'False'; ExternalWritable := 'False'} : Struct   // Opsomming van alle storingen
         A001 : Bool;   // Beveiliging aangesproken
         A002 : Bool;   // Storing detectiepunt
         A003 : Bool;   // Beveiliging klimaatregeling wegkantkast aangesproken
         A004 : Bool;   // Overspanningsbeveiliging aangesproken
      END_STRUCT;
   END_STRUCT;
END_TYPE

TYPE "C403_VAR_IF_SOS_TYPIC"
   STRUCT
      EXT_HW { ExternalAccessible := 'False'; ExternalVisible := 'False'; ExternalWritable := 'False'} : Bool;   // Sturings hardware (PLC) in storing
      STO { ExternalAccessible := 'False'; ExternalVisible := 'False'; ExternalWritable := 'False'} : Struct   // Opsomming van alle storingen
         A001 : Bool;   // Beveiliging aangesproken
         A002 : Bool;   // SOS-detectie is over 60 m tot 150 m uitgevallen
         A003 : Bool;   // SOS-detectie is over meer dan 150 m uitgevallen
      END_STRUCT;
   END_STRUCT;
END_TYPE

TYPE "C403_VAR_LVE_TYPIC"
   STRUCT
      BSC { ExternalAccessible := 'False'; ExternalVisible := 'False'; ExternalWritable := 'False'} : USInt;   // Beschikbaarheid
      STS_NEG { ExternalAccessible := 'False'; ExternalVisible := 'False'; ExternalWritable := 'False'} : USInt;   // Spookrijder gedetecteerd
      OBS { ExternalAccessible := 'False'; ExternalVisible := 'False'; ExternalWritable := 'False'} : USInt;   // Observeerbaarheid
      SIG_AV01 { ExternalAccessible := 'False'; ExternalVisible := 'False'; ExternalWritable := 'False'} : USInt;   // Signalering Stilstand gedetecteerd actief
      SIG_AV02 { ExternalAccessible := 'False'; ExternalVisible := 'False'; ExternalWritable := 'False'} : USInt;   // Signalering Snelheidsonderschrijding actief
      POS { ExternalAccessible := 'False'; ExternalVisible := 'False'; ExternalWritable := 'False'} : Bool;   // Positie van het detectiepunt
   END_STRUCT;
END_TYPE

TYPE "C406_STU_IF_CAD_TYPIC"
   STRUCT
      CMD_TOE { ExternalAccessible := 'False'; ExternalVisible := 'False'; ExternalWritable := 'False'} : Bool;   // Aansturing calamiteitendoorsteek Dicht
      CMD_OPEN { ExternalAccessible := 'False'; ExternalVisible := 'False'; ExternalWritable := 'False'} : Bool;   // Aansturing calamiteitendoorsteek Open
      CMD_RES { ExternalAccessible := 'False'; ExternalVisible := 'False'; ExternalWritable := 'False'} : Bool;   // Reset van de latched storingen
      CMD_SNS_RES { ExternalAccessible := 'False'; ExternalVisible := 'False'; ExternalWritable := 'False'} : Bool;   // Reset van de noodstop storingen
   END_STRUCT;
END_TYPE

TYPE "C406_VAR_CAD_TYPIC"
   STRUCT
      POS_STS { ExternalAccessible := 'False'; ExternalVisible := 'False'; ExternalWritable := 'False'} : USInt;   // Stand van de calamiteitendoorsteek
      BST { ExternalAccessible := 'False'; ExternalVisible := 'False'; ExternalWritable := 'False'} : USInt;   // Bestuurbaarheid
   END_STRUCT;
END_TYPE

TYPE "C406_VAR_IF_CAD_TYPIC"
   STRUCT
      BMO_HAND { ExternalAccessible := 'False'; ExternalVisible := 'False'; ExternalWritable := 'False'} : Bool;   // TRUE = CaDo in hand geschakeld FALSE = niet in hand
      STS_BEZ_TOE { ExternalAccessible := 'False'; ExternalVisible := 'False'; ExternalWritable := 'False'} : Bool;   // TRUE = Calamiteitendoorsteek bezig met beweging sluiten
      STS_BEZ_OPEN { ExternalAccessible := 'False'; ExternalVisible := 'False'; ExternalWritable := 'False'} : Bool;   // TRUE = Calamiteitendoorsteek bezig met beweging openen
      STS_POS_TOE { ExternalAccessible := 'False'; ExternalVisible := 'False'; ExternalWritable := 'False'} : Bool;   // TRUE = Calamiteitendoorsteek op stand Dicht
      STS_POS_OPEN { ExternalAccessible := 'False'; ExternalVisible := 'False'; ExternalWritable := 'False'} : Bool;   // TRUE = Calamiteitendoorsteek op stand Open
      STS_STOP { ExternalAccessible := 'False'; ExternalVisible := 'False'; ExternalWritable := 'False'} : Bool;   // TRUE = Calamiteitendoorsteek niet op een eindpositie en niet in beweging
      EXT_AUT { ExternalAccessible := 'False'; ExternalVisible := 'False'; ExternalWritable := 'False'} : Bool;   // Externe (hoofd) beveiliging aangesproken
      EXT_HW { ExternalAccessible := 'False'; ExternalVisible := 'False'; ExternalWritable := 'False'} : Bool;   // Sturings hardware (PLC) in storing
      STO { ExternalAccessible := 'False'; ExternalVisible := 'False'; ExternalWritable := 'False'} : Struct   // Opsomming van alle storingen en meldingen
         A001 : Bool;   // Beveiliging aangesproken
         A002 : Bool;   // Noodstop van de calamiteitendoorsteek is geactiveerd
         A003 : Bool;   // Storing calamiteitendoorsteek
         A004 : Bool;   // Algemene storing calamiteitendoorsteek
         A005 : Bool;   // Communicatie uitgevallen
         AT01 : Bool;   // Terugmelding Open niet tijdig bereikt
         AT02 : Bool;   // Terugmelding Dicht niet tijdig bereikt
         AT03 : Bool;   // Terugmeldingen Open en Dicht tegelijkertijd
         M001 : Bool;   // De calamiteitendoorsteek is afgekoppeld via de werkschakelaar
      END_STRUCT;
   END_STRUCT;
END_TYPE

TYPE "C501_STU_DME_TYPIC"
   STRUCT
      VGV_L { ExternalAccessible := 'False'; ExternalVisible := 'False'; ExternalWritable := 'False'} : USInt;   // Vrijgave detectie druk te laag
   END_STRUCT;
END_TYPE

TYPE "C501_STU_IF_ABP_TYPIC"
   STRUCT
      CMD { ExternalAccessible := 'False'; ExternalVisible := 'False'; ExternalWritable := 'False'} : Bool;   // Aansturing pomp (TRUE = Aan / FALSE = Uit)
      CMD_SNE { ExternalAccessible := 'False'; ExternalVisible := 'False'; ExternalWritable := 'False'} : Real;   // Sturing snelheid pomp
      LCK_AAN { ExternalAccessible := 'False'; ExternalVisible := 'False'; ExternalWritable := 'False'} : Bool;   // TRUE = Vergrendelen pomp (ook in manueel en hand)
      CMD_RES { ExternalAccessible := 'False'; ExternalVisible := 'False'; ExternalWritable := 'False'} : Bool;   // Reset van de latched storingen
   END_STRUCT;
END_TYPE

TYPE "C501_STU_IF_BBI_TYPIC"
   STRUCT
      WRE { ExternalAccessible := 'False'; ExternalVisible := 'False'; ExternalWritable := 'False'} : USInt;   // Actueel actief regime
   END_STRUCT;
END_TYPE

TYPE "C501_STU_IF_BBP_TYPIC"
   STRUCT
      CMD { ExternalAccessible := 'False'; ExternalVisible := 'False'; ExternalWritable := 'False'} : Bool;   // Aansturing pomp (TRUE = Aan / FALSE = Uit)
      LCK_AAN { ExternalAccessible := 'False'; ExternalVisible := 'False'; ExternalWritable := 'False'} : Bool;   // TRUE = Vergrendelen pomp (ook in manueel en hand)
      CMD_RES { ExternalAccessible := 'False'; ExternalVisible := 'False'; ExternalWritable := 'False'} : Bool;   // Reset van de latched storingen
   END_STRUCT;
END_TYPE

TYPE "C501_STU_IF_JKP_TYPIC"
   STRUCT
      CMD { ExternalAccessible := 'False'; ExternalVisible := 'False'; ExternalWritable := 'False'} : Bool;   // Aansturing pomp (TRUE = Aan / FALSE = Uit)
      CMD_RES { ExternalAccessible := 'False'; ExternalVisible := 'False'; ExternalWritable := 'False'} : Bool;   // Reset van de latched storingen
   END_STRUCT;
END_TYPE

TYPE "C501_STU_IF_KLG_TYPIC"
   STRUCT
      CMD { ExternalAccessible := 'False'; ExternalVisible := 'False'; ExternalWritable := 'False'} : Bool;   // Aansturing klep (TRUE = Open / FALSE = Toe)
      CMD_RES { ExternalAccessible := 'False'; ExternalVisible := 'False'; ExternalWritable := 'False'} : Bool;   // Reset van de latched storingen
   END_STRUCT;
END_TYPE

TYPE "C501_STU_JKP_TYPIC"
   STRUCT
      CMD { ExternalAccessible := 'False'; ExternalVisible := 'False'; ExternalWritable := 'False'} : USInt;   // Sturing pomp
      VGV_AAN { ExternalAccessible := 'False'; ExternalVisible := 'False'; ExternalWritable := 'False'} : USInt;   // Vrijgave aansturen pomp
   END_STRUCT;
END_TYPE

TYPE "C501_STU_JPP_TYPIC"
   STRUCT
      CMD { ExternalAccessible := 'False'; ExternalVisible := 'False'; ExternalWritable := 'False'} : USInt;   // Sturing pomppaar
      VGV_LDE { ExternalAccessible := 'False'; ExternalVisible := 'False'; ExternalWritable := 'False'} : USInt;   // Vrijgave lekdetectie
      VGV_SME_L { ExternalAccessible := 'False'; ExternalVisible := 'False'; ExternalWritable := 'False'} : USInt;   // Vrijgave detectie debiet te laag
   END_STRUCT;
END_TYPE

TYPE "C501_STU_KLG_TYPIC"
   STRUCT
      CMD { ExternalAccessible := 'False'; ExternalVisible := 'False'; ExternalWritable := 'False'} : USInt;   // Sturing klep
   END_STRUCT;
END_TYPE

TYPE "C501_STU_NME_TYPIC"
   STRUCT
      OBS { ExternalAccessible := 'False'; ExternalVisible := 'False'; ExternalWritable := 'False'} : USInt;   // Niveaumeting in of uit dienst zetten
   END_STRUCT;
END_TYPE

TYPE "C501_STU_PMP_TYPIC"
   STRUCT
      CMD { ExternalAccessible := 'False'; ExternalVisible := 'False'; ExternalWritable := 'False'} : USInt;   // Sturing pomp
      LCK_AAN { ExternalAccessible := 'False'; ExternalVisible := 'False'; ExternalWritable := 'False'} : Bool;   // TRUE = Vergrendelen pomp (ook in manueel en hand)
      CMD_SNE { ExternalAccessible := 'False'; ExternalVisible := 'False'; ExternalWritable := 'False'} : Real;   // Sturing snelheid pomp
   END_STRUCT;
END_TYPE

TYPE "C501_STU_PPP_TYPIC"
   STRUCT
      CMD { ExternalAccessible := 'False'; ExternalVisible := 'False'; ExternalWritable := 'False'} : USInt;   // Sturing pomp
      CMD_SNE { ExternalAccessible := 'False'; ExternalVisible := 'False'; ExternalWritable := 'False'} : Real;   // Sturing snelheid pomp
   END_STRUCT;
END_TYPE

TYPE "C501_STU_SME_TYPIC"
   STRUCT
      VGV_L { ExternalAccessible := 'False'; ExternalVisible := 'False'; ExternalWritable := 'False'} : USInt;   // Vrijgave detectie debiet te laag
   END_STRUCT;
END_TYPE

TYPE "C501_STU_TME_TYPIC"
   STRUCT
      VGV_L { ExternalAccessible := 'False'; ExternalVisible := 'False'; ExternalWritable := 'False'} : USInt;   // Vrijgave detectie temperatuur te laag
   END_STRUCT;
END_TYPE

TYPE "C501_VAR_BWR_TYPIC"
   STRUCT
      BSC { ExternalAccessible := 'False'; ExternalVisible := 'False'; ExternalWritable := 'False'} : USInt;   // Beschikbaarheidsstatus
   END_STRUCT;
END_TYPE

TYPE "C501_VAR_DME_TYPIC"
   STRUCT
      MWA { ExternalAccessible := 'False'; ExternalVisible := 'False'; ExternalWritable := 'False'} : USInt;   // Meetwaarde
      OBS { ExternalAccessible := 'False'; ExternalVisible := 'False'; ExternalWritable := 'False'} : USInt;   // Observeerbaarheid
   END_STRUCT;
END_TYPE

TYPE "C501_VAR_HYK_TYPIC"
   STRUCT
      DEU { ExternalAccessible := 'False'; ExternalVisible := 'False'; ExternalWritable := 'False'} : USInt;   // De hydrantkast in de verkeerskoker is geopend
      OBS { ExternalAccessible := 'False'; ExternalVisible := 'False'; ExternalWritable := 'False'} : USInt;   // Observeerbaarheid
   END_STRUCT;
END_TYPE

TYPE "C501_VAR_IF_ABP_TYPIC"
   STRUCT
      STS_AAN { ExternalAccessible := 'False'; ExternalVisible := 'False'; ExternalWritable := 'False'} : Bool;   // Pomp draait
      STS_SNE { ExternalAccessible := 'False'; ExternalVisible := 'False'; ExternalWritable := 'False'} : Real;   // Actuele snelheid pomp
      BMO_HAND { ExternalAccessible := 'False'; ExternalVisible := 'False'; ExternalWritable := 'False'} : Bool;   // Pomp in hand geschakeld
      TYD_TOT_AAN { ExternalAccessible := 'False'; ExternalVisible := 'False'; ExternalWritable := 'False'} : LInt;   // Totaal aantal draaiuren (in seconden)
      TYD_TOT_AAN_UUR { ExternalAccessible := 'False'; ExternalVisible := 'False'; ExternalWritable := 'False'} : LInt;   // Totaal aantal draaiuren (in uren)
      TYD_AAN { ExternalAccessible := 'False'; ExternalVisible := 'False'; ExternalWritable := 'False'} : Int;   // Aantal seconden dat pomp aangeschakeld is
      TYD_UIT { ExternalAccessible := 'False'; ExternalVisible := 'False'; ExternalWritable := 'False'} : Int;   // Aantal seconden dat pomp uitgeschakeld is
      ENE_MWA1 { ExternalAccessible := 'False'; ExternalVisible := 'False'; ExternalWritable := 'False'} : Real;   // Stroommeting fase 1
      ENE_MWA2 { ExternalAccessible := 'False'; ExternalVisible := 'False'; ExternalWritable := 'False'} : Real;   // Stroommeting fase 2
      ENE_MWA3 { ExternalAccessible := 'False'; ExternalVisible := 'False'; ExternalWritable := 'False'} : Real;   // Stroommeting fase 3
      EXT_HW { ExternalAccessible := 'False'; ExternalVisible := 'False'; ExternalWritable := 'False'} : Bool;   // Sturings hardware (PLC) in storing
      STO { ExternalAccessible := 'False'; ExternalVisible := 'False'; ExternalWritable := 'False'} : Struct   // Opsomming van alle storingen
         A001 : Bool;   // Beveiliging aangesproken
         A002 : Bool;   // Storing van de motorbeveiliging van de pomp
         A003 : Bool;   // Storing Frequentieomvormer
         A004 : Bool;   // Te hoge temperatuur in de motorwikkelingen
         A005 : Bool;   // De pomp is in onbalans
         A006 : Bool;   // Motorlade uitgeschakeld
         A007 : Bool;   // Motorlade in test
         A008 : Bool;   // Motorlade uitgereden
         A009 : Bool;   // Fout stroommeting fase 1
         A010 : Bool;   // Fout stroommeting fase 2
         A011 : Bool;   // Fout stroommeting fase 3
         A012 : Bool;   // Filter vervuild
         AT01 : Bool;   // Discordantie motor: terugmelding niet ontvangen
         AT02 : Bool;   // Discordantie motor: terugmelding blijft aanwezig
         M001 : Bool;   // Werkschakelaar uitgeschakeld
         M002 : Bool;   // Melding: Pomp heeft te lang niet gedraaid. Periodiek onderhoud nodig
         M003 : Bool;   // Melding: Draaitijd overschrijding
      END_STRUCT;
   END_STRUCT;
END_TYPE

TYPE "C501_VAR_IF_BBI_TYPIC"
   STRUCT
      REQ_UIT { ExternalAccessible := 'False'; ExternalVisible := 'False'; ExternalWritable := 'False'} : Bool;   // Aanvraag om regime Uit te activeren
      REQ_BWK { ExternalAccessible := 'False'; ExternalVisible := 'False'; ExternalWritable := 'False'} : Bool;   // Aanvraag om regime Bewaken te activeren
      REQ_BLUS1 { ExternalAccessible := 'False'; ExternalVisible := 'False'; ExternalWritable := 'False'} : Bool;   // Aanvraag om regime Blussen Hydrant te activeren
      REQ_BLUS2 { ExternalAccessible := 'False'; ExternalVisible := 'False'; ExternalWritable := 'False'} : Bool;   // Aanvraag om regime Blussen Hydrant en WMS te activeren
      REQ_TEST { ExternalAccessible := 'False'; ExternalVisible := 'False'; ExternalWritable := 'False'} : Bool;   // Aanvraag om regime Testen te activeren
      EXT_HW { ExternalAccessible := 'False'; ExternalVisible := 'False'; ExternalWritable := 'False'} : Bool;   // Sturings hardware (PLC) in storing
      STO { ExternalAccessible := 'False'; ExternalVisible := 'False'; ExternalWritable := 'False'} : Struct   // Opsomming van alle storingen
         A001 : Bool;   // Beveiliging aangesproken
         A002 : Bool;   // Beveiliging No-Break aangesproken
         A003 : Bool;   // Schuif ALSB uitgeschakeld
         A004 : Bool;   // Schuif ALSB in test
         A005 : Bool;   // Schuif ALSB uitgereden
         A006 : Bool;   // Lekdetectie in pomplokaal
         A007 : Bool;   // Overspanningsbeveiliging aangesproken
         A008 : Bool;   // Beveiliging kastklimatisatie aangesproken
         A009 : Bool;   // Lastscheider niet aan
      END_STRUCT;
   END_STRUCT;
END_TYPE

TYPE "C501_VAR_IF_BBP_TYPIC"
   STRUCT
      STS_AAN { ExternalAccessible := 'False'; ExternalVisible := 'False'; ExternalWritable := 'False'} : Bool;   // Pomp draait
      BMO_HAND { ExternalAccessible := 'False'; ExternalVisible := 'False'; ExternalWritable := 'False'} : Bool;   // Pomp in hand geschakeld
      TYD_TOT_AAN { ExternalAccessible := 'False'; ExternalVisible := 'False'; ExternalWritable := 'False'} : LInt;   // Totaal aantal draaiuren (in seconden)
      TYD_TOT_AAN_UUR { ExternalAccessible := 'False'; ExternalVisible := 'False'; ExternalWritable := 'False'} : LInt;   // Totaal aantal draaiuren (in uren)
      TYD_AAN { ExternalAccessible := 'False'; ExternalVisible := 'False'; ExternalWritable := 'False'} : Int;   // Aantal seconden dat pomp aangeschakeld is
      TYD_UIT { ExternalAccessible := 'False'; ExternalVisible := 'False'; ExternalWritable := 'False'} : Int;   // Aantal seconden dat pomp uitgeschakeld is
      ENE_MWA1 { ExternalAccessible := 'False'; ExternalVisible := 'False'; ExternalWritable := 'False'} : Real;   // Stroommeting fase 1
      ENE_MWA2 { ExternalAccessible := 'False'; ExternalVisible := 'False'; ExternalWritable := 'False'} : Real;   // Stroommeting fase 2
      ENE_MWA3 { ExternalAccessible := 'False'; ExternalVisible := 'False'; ExternalWritable := 'False'} : Real;   // Stroommeting fase 3
      EXT_HW { ExternalAccessible := 'False'; ExternalVisible := 'False'; ExternalWritable := 'False'} : Bool;   // Sturings hardware (PLC) in storing
      STO { ExternalAccessible := 'False'; ExternalVisible := 'False'; ExternalWritable := 'False'} : Struct   // Opsomming van alle storingen
         A001 : Bool;   // Beveiliging aangesproken
         A002 : Bool;   // Storing van de motorbeveiliging van de pomp
         A003 : Bool;   // Storing softstarter
         A004 : Bool;   // Te hoge temperatuur in de motorwikkelingen
         A005 : Bool;   // De pomp is in onbalans
         A006 : Bool;   // Motorlade uitgeschakeld
         A007 : Bool;   // Motorlade in test
         A008 : Bool;   // Motorlade uitgereden
         A009 : Bool;   // Fout stroommeting fase 1
         A010 : Bool;   // Fout stroommeting fase 2
         A011 : Bool;   // Fout stroommeting fase 3
         A012 : Bool;   // Filter vervuild
         AT01 : Bool;   // Discordantie motor: terugmelding niet ontvangen
         AT02 : Bool;   // Discordantie motor: terugmelding blijft aanwezig
         M001 : Bool;   // Werkschakelaar uitgeschakeld
         M002 : Bool;   // Melding: Pomp heeft te lang niet gedraaid. Periodiek onderhoud nodig
         M003 : Bool;   // Melding: Draaitijd overschrijding
      END_STRUCT;
   END_STRUCT;
END_TYPE

TYPE "C501_VAR_IF_DME_TYPIC"
   STRUCT
      MWA { ExternalAccessible := 'False'; ExternalVisible := 'False'; ExternalWritable := 'False'} : Real;   // Meetwaarde
      EXT_HW { ExternalAccessible := 'False'; ExternalVisible := 'False'; ExternalWritable := 'False'} : Bool;   // Sturings hardware (PLC) in storing
      STO { ExternalAccessible := 'False'; ExternalVisible := 'False'; ExternalWritable := 'False'} : Struct   // Opsomming van alle storingen
         A001 : Bool;   // Beveiliging aangesproken
         A002 : Bool;   // Draadbreuk analoge meting
         A003 : Bool;   // Meetbereik overschreden
         A004 : Bool;   // Drukmeter geeft storing
      END_STRUCT;
   END_STRUCT;
END_TYPE

TYPE "C501_VAR_IF_HYK_TYPIC"
   STRUCT
      DEC { ExternalAccessible := 'False'; ExternalVisible := 'False'; ExternalWritable := 'False'} : Bool;   // De hydrantkast in de verkeerskoker is gesloten
      EXT_HW { ExternalAccessible := 'False'; ExternalVisible := 'False'; ExternalWritable := 'False'} : Bool;   // Sturings hardware (PLC) in storing
      STO { ExternalAccessible := 'False'; ExternalVisible := 'False'; ExternalWritable := 'False'} : Struct   // Opsomming van alle storingen
         A001 : Bool;   // Beveiliging aangesproken
         A002 : Bool;   // Temperatuur te laag
      END_STRUCT;
   END_STRUCT;
END_TYPE

TYPE "C501_VAR_IF_JKP_TYPIC"
   STRUCT
      STS_AAN { ExternalAccessible := 'False'; ExternalVisible := 'False'; ExternalWritable := 'False'} : Bool;   // Pomp draait
      BMO_HAND { ExternalAccessible := 'False'; ExternalVisible := 'False'; ExternalWritable := 'False'} : Bool;   // Pomp in hand geschakeld
      TYD_TOT_AAN { ExternalAccessible := 'False'; ExternalVisible := 'False'; ExternalWritable := 'False'} : LInt;   // Totaal aantal draaiuren in seconden
      TYD_TOT_AAN_UUR { ExternalAccessible := 'False'; ExternalVisible := 'False'; ExternalWritable := 'False'} : LInt;   // Totaal aantal draaiuren (in uren)
      TYD_AAN { ExternalAccessible := 'False'; ExternalVisible := 'False'; ExternalWritable := 'False'} : Int;   // Aantal seconden dat pomp aangeschakeld is
      TYD_UIT { ExternalAccessible := 'False'; ExternalVisible := 'False'; ExternalWritable := 'False'} : Int;   // Aantal seconden dat pomp uitgeschakeld is
      EXT_HW { ExternalAccessible := 'False'; ExternalVisible := 'False'; ExternalWritable := 'False'} : Bool;   // Sturings hardware (PLC) in storing
      STO { ExternalAccessible := 'False'; ExternalVisible := 'False'; ExternalWritable := 'False'} : Struct   // Opsomming van alle storingen
         A001 : Bool;   // Beveiliging aangesproken
         A002 : Bool;   // Filter vervuild
         A003 : Bool;   // Storing van de motorbeveiliging van de pomp
         AT01 : Bool;   // Discordantie motor: terugmelding niet ontvangen
         AT02 : Bool;   // Discordantie motor: terugmelding blijft aanwezig
         M001 : Bool;   // Werkschakelaar uitgeschakeld
         M002 : Bool;   // Melding: Pomp heeft te lang niet gedraaid. Periodiek onderhoud nodig
      END_STRUCT;
   END_STRUCT;
END_TYPE

TYPE "C501_VAR_IF_KLG_TYPIC"
   STRUCT
      STS_OPEN { ExternalAccessible := 'False'; ExternalVisible := 'False'; ExternalWritable := 'False'} : Bool;   // Motorgestuurde klep is open
      STS_TOE { ExternalAccessible := 'False'; ExternalVisible := 'False'; ExternalWritable := 'False'} : Bool;   // Motorgestuurde klep is toe
      STS_BEZ_OPEN { ExternalAccessible := 'False'; ExternalVisible := 'False'; ExternalWritable := 'False'} : Bool;   // Motorgestuurde klep is aan het openen (1 = Open)
      STS_BEZ_TOE { ExternalAccessible := 'False'; ExternalVisible := 'False'; ExternalWritable := 'False'} : Bool;   // Motorgestuurde klep is aan het sluiten (1 = Toe)
      BMO_HAND { ExternalAccessible := 'False'; ExternalVisible := 'False'; ExternalWritable := 'False'} : Bool;   // TRUE = in hand geschakeld FALSE = niet in hand
      EXT_HW { ExternalAccessible := 'False'; ExternalVisible := 'False'; ExternalWritable := 'False'} : Bool;   // Sturings hardware (PLC) in storing
      STO { ExternalAccessible := 'False'; ExternalVisible := 'False'; ExternalWritable := 'False'} : Struct   // Opsomming van alle storingen
         A001 : Bool;   // Beveiliging aangesproken
         AT01 : Bool;   // Terugmelding Open niet ontvangen
         AT02 : Bool;   // Terugmelding Dicht niet ontvangen
         AT03 : Bool;   // Terugmeldingen Open en Dicht tegelijkertijd
      END_STRUCT;
   END_STRUCT;
END_TYPE

TYPE "C501_VAR_IF_KLH_TYPIC"
   STRUCT
      STS_OPEN { ExternalAccessible := 'False'; ExternalVisible := 'False'; ExternalWritable := 'False'} : Bool;   // Handbediende klep is open
      STS_TOE { ExternalAccessible := 'False'; ExternalVisible := 'False'; ExternalWritable := 'False'} : Bool;   // Handbediende klep is toe
      EXT_HW { ExternalAccessible := 'False'; ExternalVisible := 'False'; ExternalWritable := 'False'} : Bool;   // Sturings hardware (PLC) in storing
      STO { ExternalAccessible := 'False'; ExternalVisible := 'False'; ExternalWritable := 'False'} : Struct   // Opsomming van alle storingen
         A001 : Bool;   // Terugmeldingen Open en Dicht tegelijk
      END_STRUCT;
   END_STRUCT;
END_TYPE

TYPE "C501_VAR_IF_NME_TYPIC"
   STRUCT
      MWA { ExternalAccessible := 'False'; ExternalVisible := 'False'; ExternalWritable := 'False'} : Real;   // Meetwaarde
      HW { ExternalAccessible := 'False'; ExternalVisible := 'False'; ExternalWritable := 'False'} : USInt;   // Hoogwater vlotter
      VHW { ExternalAccessible := 'False'; ExternalVisible := 'False'; ExternalWritable := 'False'} : USInt;   // Voorwaarschuwing hoogwater
      SD { ExternalAccessible := 'False'; ExternalVisible := 'False'; ExternalWritable := 'False'} : USInt;   // Suppletie dicht
      SO { ExternalAccessible := 'False'; ExternalVisible := 'False'; ExternalWritable := 'False'} : USInt;   // Suppletie open
      VRL { ExternalAccessible := 'False'; ExternalVisible := 'False'; ExternalWritable := 'False'} : USInt;   // Voorwaarschuwing reservoir leeg
      RL { ExternalAccessible := 'False'; ExternalVisible := 'False'; ExternalWritable := 'False'} : USInt;   // Reservoir leeg
      EXT_HW { ExternalAccessible := 'False'; ExternalVisible := 'False'; ExternalWritable := 'False'} : Bool;   // Sturings hardware (PLC) in storing
      STO { ExternalAccessible := 'False'; ExternalVisible := 'False'; ExternalWritable := 'False'} : Struct   // Opsomming van alle storingen
         A001 : Bool;   // Beveiliging aangesproken
         A002 : Bool;   // Draadbreuk analoge meting
         A003 : Bool;   // Meetbereik overschreden
         A004 : Bool;   // Status vlotters inconsistent
      END_STRUCT;
   END_STRUCT;
END_TYPE

TYPE "C501_VAR_IF_SME_TYPIC"
   STRUCT
      MWA { ExternalAccessible := 'False'; ExternalVisible := 'False'; ExternalWritable := 'False'} : Real;   // Meetwaarde
      EXT_HW { ExternalAccessible := 'False'; ExternalVisible := 'False'; ExternalWritable := 'False'} : Bool;   // Sturings hardware (PLC) in storing
      STO { ExternalAccessible := 'False'; ExternalVisible := 'False'; ExternalWritable := 'False'} : Struct   // Opsomming van alle storingen
         A001 : Bool;   // Beveiliging aangesproken
         A002 : Bool;   // Draadbreuk analoge meting
         A003 : Bool;   // Meetbereik overschreden
         A004 : Bool;   // Debietmeter geeft storing
      END_STRUCT;
   END_STRUCT;
END_TYPE

TYPE "C501_VAR_IF_TME_TYPIC"
   STRUCT
      MWA { ExternalAccessible := 'False'; ExternalVisible := 'False'; ExternalWritable := 'False'} : Real;   // Meetwaarde
      EXT_HW { ExternalAccessible := 'False'; ExternalVisible := 'False'; ExternalWritable := 'False'} : Bool;   // Sturings hardware (PLC) in storing
      STO { ExternalAccessible := 'False'; ExternalVisible := 'False'; ExternalWritable := 'False'} : Struct   // Opsomming van alle storingen
         A001 : Bool;   // Beveiliging aangesproken
         A002 : Bool;   // Draadbreuk analoge meting
         A003 : Bool;   // Meetbereik overschreden
         A004 : Bool;   // Temperatuurmeter geeft storing
      END_STRUCT;
   END_STRUCT;
END_TYPE

TYPE "C501_VAR_IF_TRA_TYPIC"
   STRUCT
      EXT_HW { ExternalAccessible := 'False'; ExternalVisible := 'False'; ExternalWritable := 'False'} : Bool;   // Sturings hardware (PLC) in storing
      STO { ExternalAccessible := 'False'; ExternalVisible := 'False'; ExternalWritable := 'False'} : Struct   // Opsomming van alle storingen
         A001 : Bool;   // Storing vorstbeveiliging
      END_STRUCT;
   END_STRUCT;
END_TYPE

TYPE "C501_VAR_JKP_TYPIC"
   STRUCT
      STS { ExternalAccessible := 'False'; ExternalVisible := 'False'; ExternalWritable := 'False'} : USInt;   // Status van de pomp
      BMO { ExternalAccessible := 'False'; ExternalVisible := 'False'; ExternalWritable := 'False'} : USInt;   // Bedieningsmode
      BST { ExternalAccessible := 'False'; ExternalVisible := 'False'; ExternalWritable := 'False'} : USInt;   // Bestuurbaarheid
      PWR { ExternalAccessible := 'False'; ExternalVisible := 'False'; ExternalWritable := 'False'} : Real;   // Actueel vermogen van de pomp
      TYD_TOT_AAN { ExternalAccessible := 'False'; ExternalVisible := 'False'; ExternalWritable := 'False'} : LInt;   // Totaal aantal draaiuren
      TYD_AAN { ExternalAccessible := 'False'; ExternalVisible := 'False'; ExternalWritable := 'False'} : Int;   // Tijdsduur dat pomp aangeschakeld is
      TYD_UIT { ExternalAccessible := 'False'; ExternalVisible := 'False'; ExternalWritable := 'False'} : Int;   // Tijdsduur dat pomp uitgeschakeld is
   END_STRUCT;
END_TYPE

TYPE "C501_VAR_JPP_TYPIC"
   STRUCT
      BST { ExternalAccessible := 'False'; ExternalVisible := 'False'; ExternalWritable := 'False'} : USInt;   // Bestuurbaarheid
      BSC { ExternalAccessible := 'False'; ExternalVisible := 'False'; ExternalWritable := 'False'} : USInt;   // NOK = Storing aanwezig die beschikbaarheid beinvloed
      PWR { ExternalAccessible := 'False'; ExternalVisible := 'False'; ExternalWritable := 'False'} : Real;   // Actueel vermogen van het pomppaar
      STS { ExternalAccessible := 'False'; ExternalVisible := 'False'; ExternalWritable := 'False'} : USInt;   // Aan = er is minstens een jockeypomp aangeschakeld Uit = alle jockeypompen zijn uit
   END_STRUCT;
END_TYPE

TYPE "C501_VAR_KLG_TYPIC"
   STRUCT
      STS { ExternalAccessible := 'False'; ExternalVisible := 'False'; ExternalWritable := 'False'} : USInt;   // Status van de klep
      BMO { ExternalAccessible := 'False'; ExternalVisible := 'False'; ExternalWritable := 'False'} : USInt;   // Bedieningsmode
      BST { ExternalAccessible := 'False'; ExternalVisible := 'False'; ExternalWritable := 'False'} : USInt;   // Bestuurbaarheid
   END_STRUCT;
END_TYPE

TYPE "C501_VAR_KLH_TYPIC"
   STRUCT
      OBS { ExternalAccessible := 'False'; ExternalVisible := 'False'; ExternalWritable := 'False'} : USInt;   // Observeerbaarheid
      VAR_STS_NORM { ExternalAccessible := 'False'; ExternalVisible := 'False'; ExternalWritable := 'False'} : USInt;   // Ja = Klep in normale positie Nee = Niet in normale positie
      VAR_BSC { ExternalAccessible := 'False'; ExternalVisible := 'False'; ExternalWritable := 'False'} : USInt;   // Ja = Brandblusinstallatie onbeschikbaar als niet in normaal Nee = Brandblusinstallatie wordt niet onbeschikbaar
   END_STRUCT;
END_TYPE

TYPE "C501_VAR_NME_TYPIC"
   STRUCT
      MWA { ExternalAccessible := 'False'; ExternalVisible := 'False'; ExternalWritable := 'False'} : Real;   // Meetwaarde
      STS_HW { ExternalAccessible := 'False'; ExternalVisible := 'False'; ExternalWritable := 'False'} : USInt;   // Hoogwater vlotter
      STS_VHW { ExternalAccessible := 'False'; ExternalVisible := 'False'; ExternalWritable := 'False'} : USInt;   // Voorwaarschuwing hoogwater
      STS_SD { ExternalAccessible := 'False'; ExternalVisible := 'False'; ExternalWritable := 'False'} : USInt;   // Suppletie dicht
      STS_SO { ExternalAccessible := 'False'; ExternalVisible := 'False'; ExternalWritable := 'False'} : USInt;   // Suppletie open
      STS_VRL { ExternalAccessible := 'False'; ExternalVisible := 'False'; ExternalWritable := 'False'} : USInt;   // Voorwaarschuwing reservoir leeg
      STS_RL { ExternalAccessible := 'False'; ExternalVisible := 'False'; ExternalWritable := 'False'} : USInt;   // Reservoir leeg
      OBS { ExternalAccessible := 'False'; ExternalVisible := 'False'; ExternalWritable := 'False'} : USInt;   // Observeerbaarheid
   END_STRUCT;
END_TYPE

TYPE "C501_VAR_PMP_TYPIC"
   STRUCT
      STS { ExternalAccessible := 'False'; ExternalVisible := 'False'; ExternalWritable := 'False'} : USInt;   // Status van de pomp
      BMO { ExternalAccessible := 'False'; ExternalVisible := 'False'; ExternalWritable := 'False'} : USInt;   // Bedieningsmode
      BST { ExternalAccessible := 'False'; ExternalVisible := 'False'; ExternalWritable := 'False'} : USInt;   // Bestuurbaarheid
      PWR { ExternalAccessible := 'False'; ExternalVisible := 'False'; ExternalWritable := 'False'} : Real;   // Actueel vermogen van de pomp
      TYD_TOT_AAN { ExternalAccessible := 'False'; ExternalVisible := 'False'; ExternalWritable := 'False'} : LInt;   // Totaal aantal draaiuren
      TYD_AAN { ExternalAccessible := 'False'; ExternalVisible := 'False'; ExternalWritable := 'False'} : Int;   // Tijdsduur dat pomp aangeschakeld is
      TYD_UIT { ExternalAccessible := 'False'; ExternalVisible := 'False'; ExternalWritable := 'False'} : Int;   // Tijdsduur dat pomp uitgeschakeld is
   END_STRUCT;
END_TYPE

TYPE "C501_VAR_PPP_TYPIC"
   STRUCT
      BST { ExternalAccessible := 'False'; ExternalVisible := 'False'; ExternalWritable := 'False'} : USInt;   // Bestuurbaarheid
      BSC { ExternalAccessible := 'False'; ExternalVisible := 'False'; ExternalWritable := 'False'} : USInt;   // NOK = storing aanwezig die beschikbaarheid beinvloed
      PWR { ExternalAccessible := 'False'; ExternalVisible := 'False'; ExternalWritable := 'False'} : Real;   // Actueel vermogen van het pomppaar
      STS { ExternalAccessible := 'False'; ExternalVisible := 'False'; ExternalWritable := 'False'} : USInt;   // Aan = er is minstens een pomp aangeschakeld Uit = alle pompen zijn uit
   END_STRUCT;
END_TYPE

TYPE "C501_VAR_SME_TYPIC"
   STRUCT
      MWA { ExternalAccessible := 'False'; ExternalVisible := 'False'; ExternalWritable := 'False'} : USInt;   // Meetwaarde
      OBS { ExternalAccessible := 'False'; ExternalVisible := 'False'; ExternalWritable := 'False'} : USInt;   // Observeerbaarheid
   END_STRUCT;
END_TYPE

